LIN {X 0,Y 354.832,Z 168.283,A -85,B 0,C 180,E1 -13567.896,E2 -13567.896} C_VEL
LIN {X 0,Y 354.92,Z 168.273,A -85,B 0,C 180,E1 -13571.894,E2 -13571.894} C_VEL
LIN {X 0,Y 354.941,Z 168.271,A -85,B 0,C 180,E1 -13575.983,E2 -13575.983} C_VEL
LIN {X 0,Y 354.977,Z 168.266,A -85,B 0,C 180,E1 -13579.738,E2 -13579.738} C_VEL
LIN {X 0,Y 355.114,Z 168.252,A -85,B 0,C 180,E1 -13582.039,E2 -13582.039} C_VEL
LIN {X 0,Y 355.093,Z 168.255,A -85,B 0,C 180,E1 -13584.323,E2 -13584.323} C_VEL
LIN {X 0,Y 355.245,Z 168.235,A -85,B 0,C 180,E1 -13587.734,E2 -13587.734} C_VEL
LIN {X 0,Y 355.242,Z 168.235,A -85,B 0,C 180,E1 -13592.269,E2 -13592.269} C_VEL
LIN {X 0,Y 355.141,Z 168.245,A -85,B 0,C 180,E1 -13596.821,E2 -13596.821} C_VEL
LIN {X 0,Y 355.018,Z 168.261,A -85,B 0,C 180,E1 -13599.114,E2 -13599.114} C_VEL
LIN {X 0,Y 354.924,Z 168.271,A -85,B 0,C 180,E1 -13602.582,E2 -13602.582} C_VEL
LIN {X 0,Y 354.893,Z 168.276,A -85,B 0,C 180,E1 -13606.097,E2 -13606.097} C_VEL
LIN {X 0,Y 354.905,Z 168.274,A -85,B 0,C 180,E1 -13608.474,E2 -13608.474} C_VEL
LIN {X 0,Y 354.811,Z 168.286,A -85,B 0,C 180,E1 -13612.109,E2 -13612.109} C_VEL
LIN {X 0,Y 354.804,Z 168.287,A -85,B 0,C 180,E1 -13615.836,E2 -13615.836} C_VEL
LIN {X 0,Y 354.804,Z 168.288,A -85,B 0,C 180,E1 -13619.685,E2 -13619.685} C_VEL
LIN {X 0,Y 354.792,Z 168.29,A -85,B 0,C 180,E1 -13622.335,E2 -13622.335} C_VEL
LIN {X 0,Y 354.826,Z 168.284,A -85,B 0,C 180,E1 -13625.7,E2 -13625.7} C_VEL
LIN {X 0,Y 354.773,Z 168.291,A -85,B 0,C 180,E1 -13629.413,E2 -13629.413} C_VEL
LIN {X 0,Y 354.79,Z 168.292,A -85,B 0,C 180,E1 -13632.867,E2 -13632.867} C_VEL
LIN {X 0,Y 354.772,Z 168.293,A -85,B 0,C 180,E1 -13636.104,E2 -13636.104} C_VEL
LIN {X 0,Y 354.773,Z 168.289,A -85,B 0,C 180,E1 -13639.618,E2 -13639.618} C_VEL
LIN {X 0,Y 354.806,Z 168.29,A -85,B 0,C 180,E1 -13642.405,E2 -13642.405} C_VEL
LIN {X 0,Y 354.827,Z 168.286,A -85,B 0,C 180,E1 -13644.549,E2 -13644.549} C_VEL
LIN {X 0,Y 354.259,Z 168.738,A -85,B 0,C 180,E1 -13645.493,E2 -13645.493} C_VEL
LIN {X 0,Y 352.913,Z 169.909,A -85,B 0,C 180,E1 -13646.41,E2 -13646.41} C_VEL
LIN {X 0,Y 349.778,Z 173.519,A -85,B 0,C 180,E1 -13648.211,E2 -13648.211} C_VEL
LIN {X 0,Y 348.879,Z 176.103,A -85,B 0,C 180,E1 -13649.443,E2 -13649.443} C_VEL
LIN {X 0,Y 348.478,Z 182.428,A -85,B 0,C 180,E1 -13652.548,E2 -13652.548} C_VEL
LIN {X 0,Y 347.923,Z 189.955,A -85,B 0,C 180,E1 -13656.172,E2 -13656.172} C_VEL
LIN {X 0,Y 347.454,Z 197.78,A -85,B 0,C 180,E1 -13659.888,E2 -13659.888} C_VEL
LIN {X 0,Y 347.058,Z 205.567,A -85,B 0,C 180,E1 -13663.531,E2 -13663.531} C_VEL
LIN {X 0,Y 346.795,Z 213.332,A -85,B 0,C 180,E1 -13667.119,E2 -13667.119} C_VEL
LIN {X 0,Y 346.657,Z 216.242,A -85,B 0,C 180,E1 -13668.377,E2 -13668.377} C_VEL
LIN {X 0,Y 347.531,Z 227.151,A -85,B 0,C 180,E1 -13669.071,E2 -13669.071} C_VEL
LIN {X 0,Y 348.261,Z 236.165,A -85,B 0,C 180,E1 -13669.83,E2 -13669.83} C_VEL
LIN {X 0,Y 347.759,Z 245.798,A -85,B 0,C 180,E1 -13670.843,E2 -13670.843} C_VEL
LIN {X 0,Y 347.321,Z 255.426,A -85,B 0,C 180,E1 -13672.15,E2 -13672.15} C_VEL
LIN {X 0,Y 347.005,Z 261.907,A -85,B 0,C 180,E1 -13673.258,E2 -13673.258} C_VEL
LIN {X 0,Y 346.787,Z 268.916,A -85,B 0,C 180,E1 -13674.768,E2 -13674.768} C_VEL
LIN {X 0,Y 346.59,Z 273.17,A -85,B 0,C 180,E1 -13675.93,E2 -13675.93} C_VEL
LIN {X 0,Y 346.348,Z 277.972,A -85,B 0,C 180,E1 -13677.674,E2 -13677.674} C_VEL
LIN {X 0,Y 346.339,Z 280.246,A -85,B 0,C 180,E1 -13678.837,E2 -13678.837} C_VEL
LIN {X 0,Y 346.387,Z 281.827,A -85,B 0,C 180,E1 -13680,E2 -13680} C_VEL
LIN {X 0,Y 346.491,Z 282.748,A -85,B 0,C 180,E1 -13681.162,E2 -13681.162} C_VEL
LIN {X 0,Y 346.674,Z 283.01,A -85,B 0,C 180,E1 -13682.324,E2 -13682.324} C_VEL
LIN {X 0,Y 346.972,Z 282.623,A -85,B 0,C 180,E1 -13683.484,E2 -13683.484} C_VEL
LIN {X 0,Y 347.505,Z 281.586,A -85,B 0,C 180,E1 -13684.64,E2 -13684.64} C_VEL
LIN {X 0,Y 347.852,Z 278.872,A -85,B 0,C 180,E1 -13686.38,E2 -13686.38} C_VEL
LIN {X 0,Y 348.695,Z 274.586,A -85,B 0,C 180,E1 -13688.111,E2 -13688.111} C_VEL
LIN {X 0,Y 349.806,Z 269.133,A -85,B 0,C 180,E1 -13689.678,E2 -13689.678} C_VEL
LIN {X 0,Y 351.27,Z 261.867,A -85,B 0,C 180,E1 -13691.249,E2 -13691.249} C_VEL
LIN {X 0,Y 352.727,Z 253.419,A -85,B 0,C 180,E1 -13692.661,E2 -13692.661} C_VEL
LIN {X 0,Y 353.847,Z 246.132,A -85,B 0,C 180,E1 -13693.642,E2 -13693.642} C_VEL
LIN {X 0,Y 353.083,Z 236.877,A -85,B 0,C 180,E1 -13694.849,E2 -13694.849} C_VEL
LIN {X 0,Y 351.358,Z 227.651,A -85,B 0,C 180,E1 -13695.949,E2 -13695.949} C_VEL
LIN {X 0,Y 348.627,Z 217.69,A -85,B 0,C 180,E1 -13697.072,E2 -13697.072} C_VEL
LIN {X 0,Y 349.409,Z 211.359,A -85,B 0,C 180,E1 -13700.61,E2 -13700.61} C_VEL
LIN {X 0,Y 350.246,Z 206.213,A -85,B 0,C 180,E1 -13703.661,E2 -13703.661} C_VEL
LIN {X 0,Y 351.389,Z 200.419,A -85,B 0,C 180,E1 -13707.388,E2 -13707.388} C_VEL
LIN {X 0,Y 352.288,Z 196.86,A -85,B 0,C 180,E1 -13709.917,E2 -13709.917} C_VEL
LIN {X 0,Y 352.647,Z 195.246,A -85,B 0,C 180,E1 -13711.209,E2 -13711.209} C_VEL
LIN {X 0,Y 352.835,Z 193.025,A -85,B 0,C 180,E1 -13713.217,E2 -13713.217} C_VEL
LIN {X 0,Y 352.595,Z 190.094,A -85,B 0,C 180,E1 -13716.725,E2 -13716.725} C_VEL
LIN {X 0,Y 352.358,Z 188.51,A -85,B 0,C 180,E1 -13719.662,E2 -13719.662} C_VEL
LIN {X 0,Y 352.317,Z 187.695,A -85,B 0,C 180,E1 -13722.706,E2 -13722.706} C_VEL
LIN {X 0,Y 352.457,Z 187.837,A -85,B 0,C 180,E1 -13725.877,E2 -13725.877} C_VEL
LIN {X 0,Y 352.75,Z 188.963,A -85,B 0,C 180,E1 -13728.891,E2 -13728.891} C_VEL
LIN {X 0,Y 353.2,Z 191.093,A -85,B 0,C 180,E1 -13731.913,E2 -13731.913} C_VEL
LIN {X 0,Y 353.859,Z 194.075,A -85,B 0,C 180,E1 -13734.831,E2 -13734.831} C_VEL
LIN {X 0,Y 354.621,Z 197.872,A -85,B 0,C 180,E1 -13737.648,E2 -13737.648} C_VEL
LIN {X 0,Y 355.095,Z 201.146,A -85,B 0,C 180,E1 -13739.687,E2 -13739.687} C_VEL
LIN {X 0,Y 354.861,Z 203.838,A -85,B 0,C 180,E1 -13741.084,E2 -13741.084} C_VEL
LIN {X 0,Y 352.926,Z 210.525,A -85,B 0,C 180,E1 -13744.016,E2 -13744.016} C_VEL
LIN {X 0,Y 350.745,Z 220.327,A -85,B 0,C 180,E1 -13747.931,E2 -13747.931} C_VEL
LIN {X 0,Y 353.911,Z 233.578,A -85,B 0,C 180,E1 -13748.961,E2 -13748.961} C_VEL
LIN {X 0,Y 355.2,Z 243.511,A -85,B 0,C 180,E1 -13749.771,E2 -13749.771} C_VEL
LIN {X 0,Y 355.188,Z 251.982,A -85,B 0,C 180,E1 -13750.493,E2 -13750.493} C_VEL
LIN {X 0,Y 353.684,Z 263.835,A -85,B 0,C 180,E1 -13751.61,E2 -13751.61} C_VEL
LIN {X 0,Y 352.068,Z 274.487,A -85,B 0,C 180,E1 -13752.874,E2 -13752.874} C_VEL
LIN {X 0,Y 350.347,Z 284.861,A -85,B 0,C 180,E1 -13754.429,E2 -13754.429} C_VEL
LIN {X 0,Y 349.222,Z 293.327,A -85,B 0,C 180,E1 -13756.023,E2 -13756.023} C_VEL
LIN {X 0,Y 348.027,Z 300.772,A -85,B 0,C 180,E1 -13757.757,E2 -13757.757} C_VEL
LIN {X 0,Y 347.198,Z 306.772,A -85,B 0,C 180,E1 -13759.502,E2 -13759.502} C_VEL
LIN {X 0,Y 346.647,Z 311.533,A -85,B 0,C 180,E1 -13761.252,E2 -13761.252} C_VEL
LIN {X 0,Y 346.342,Z 315.161,A -85,B 0,C 180,E1 -13763.005,E2 -13763.005} C_VEL
LIN {X 0,Y 346.251,Z 316.986,A -85,B 0,C 180,E1 -13764.173,E2 -13764.173} C_VEL
LIN {X 0,Y 346.215,Z 318.385,A -85,B 0,C 180,E1 -13765.341,E2 -13765.341} C_VEL
LIN {X 0,Y 346.197,Z 319.375,A -85,B 0,C 180,E1 -13766.507,E2 -13766.507} C_VEL
LIN {X 0,Y 346.245,Z 319.9,A -85,B 0,C 180,E1 -13767.672,E2 -13767.672} C_VEL
LIN {X 0,Y 346.385,Z 320.016,A -85,B 0,C 180,E1 -13768.836,E2 -13768.836} C_VEL
LIN {X 0,Y 346.394,Z 319.713,A -85,B 0,C 180,E1 -13769.998,E2 -13769.998} C_VEL
LIN {X 0,Y 346.419,Z 318.933,A -85,B 0,C 180,E1 -13771.161,E2 -13771.161} C_VEL
LIN {X 0,Y 346.459,Z 317.723,A -85,B 0,C 180,E1 -13772.323,E2 -13772.323} C_VEL
LIN {X 0,Y 346.313,Z 315.011,A -85,B 0,C 180,E1 -13774.071,E2 -13774.071} C_VEL
LIN {X 0,Y 346.396,Z 311.191,A -85,B 0,C 180,E1 -13775.82,E2 -13775.82} C_VEL
LIN {X 0,Y 346.496,Z 306.1,A -85,B 0,C 180,E1 -13777.574,E2 -13777.574} C_VEL
LIN {X 0,Y 346.692,Z 299.54,A -85,B 0,C 180,E1 -13779.331,E2 -13779.331} C_VEL
LIN {X 0,Y 347.11,Z 291.289,A -85,B 0,C 180,E1 -13781.088,E2 -13781.088} C_VEL
LIN {X 0,Y 347.617,Z 282.661,A -85,B 0,C 180,E1 -13782.551,E2 -13782.551} C_VEL
LIN {X 0,Y 348.249,Z 273.162,A -85,B 0,C 180,E1 -13783.864,E2 -13783.864} C_VEL
LIN {X 0,Y 348.924,Z 262.248,A -85,B 0,C 180,E1 -13785.073,E2 -13785.073} C_VEL
LIN {X 0,Y 349.637,Z 251.072,A -85,B 0,C 180,E1 -13786.043,E2 -13786.043} C_VEL
LIN {X 0,Y 349.783,Z 243.763,A -85,B 0,C 180,E1 -13786.56,E2 -13786.56} C_VEL
LIN {X 0,Y 348.453,Z 230.087,A -85,B 0,C 180,E1 -13787.324,E2 -13787.324} C_VEL
LIN {X 0,Y 347.768,Z 220.166,A -85,B 0,C 180,E1 -13787.729,E2 -13787.729} C_VEL
LIN {X 0,Y 349.042,Z 206.707,A -85,B 0,C 180,E1 -13792.147,E2 -13792.147} C_VEL
LIN {X 0,Y 350.509,Z 194.632,A -85,B 0,C 180,E1 -13796.173,E2 -13796.173} C_VEL
LIN {X 0,Y 351.264,Z 188.272,A -85,B 0,C 180,E1 -13798.316,E2 -13798.316} C_VEL
LIN {X 0,Y 350.363,Z 182.502,A -85,B 0,C 180,E1 -13800.396,E2 -13800.396} C_VEL
LIN {X 0,Y 348.285,Z 171.813,A -85,B 0,C 180,E1 -13804.4,E2 -13804.4} C_VEL
LIN {X 0,Y 347.78,Z 169.17,A -85,B 0,C 180,E1 -13805.428,E2 -13805.428} C_VEL
LIN {X 0,Y 347.745,Z 169.171,A -85,B 0,C 180,E1 -13808.791,E2 -13808.791} C_VEL
LIN {X 0,Y 347.742,Z 169.166,A -85,B 0,C 180,E1 -13811.828,E2 -13811.828} C_VEL
LIN {X 0,Y 347.789,Z 169.162,A -85,B 0,C 180,E1 -13815.01,E2 -13815.01} C_VEL
LIN {X 0,Y 347.775,Z 169.167,A -85,B 0,C 180,E1 -13818.389,E2 -13818.389} C_VEL
LIN {X 0,Y 347.767,Z 169.167,A -85,B 0,C 180,E1 -13822.009,E2 -13822.009} C_VEL
LIN {X 0,Y 347.733,Z 169.168,A -85,B 0,C 180,E1 -13825.535,E2 -13825.535} C_VEL
LIN {X 0,Y 347.752,Z 169.168,A -85,B 0,C 180,E1 -13829.652,E2 -13829.652} C_VEL
LIN {X 0,Y 347.84,Z 169.154,A -85,B 0,C 180,E1 -13832.743,E2 -13832.743} C_VEL
LIN {X 0,Y 347.772,Z 169.165,A -85,B 0,C 180,E1 -13836.161,E2 -13836.161} C_VEL
LIN {X 0,Y 347.798,Z 169.163,A -85,B 0,C 180,E1 -13839.908,E2 -13839.908} C_VEL
LIN {X 0,Y 347.853,Z 169.153,A -85,B 0,C 180,E1 -13842.358,E2 -13842.358} C_VEL
LIN {X 0,Y 347.883,Z 169.15,A -85,B 0,C 180,E1 -13845.97,E2 -13845.97} C_VEL
LIN {X 0,Y 347.916,Z 169.148,A -85,B 0,C 180,E1 -13849.525,E2 -13849.525} C_VEL
LIN {X 0,Y 348.081,Z 169.128,A -85,B 0,C 180,E1 -13853.042,E2 -13853.042} C_VEL
LIN {X 0,Y 348.195,Z 169.111,A -85,B 0,C 180,E1 -13857.686,E2 -13857.686} C_VEL
LIN {X 0,Y 348.331,Z 169.093,A -85,B 0,C 180,E1 -13860,E2 -13860} C_VEL
LIN {X 0,Y 348.189,Z 169.111,A -85,B 0,C 180,E1 -13862.314,E2 -13862.314} C_VEL
LIN {X 0,Y 348.091,Z 169.127,A -85,B 0,C 180,E1 -13866.958,E2 -13866.958} C_VEL
LIN {X 0,Y 347.955,Z 169.141,A -85,B 0,C 180,E1 -13869.299,E2 -13869.299} C_VEL
LIN {X 0,Y 347.88,Z 169.152,A -85,B 0,C 180,E1 -13872.84,E2 -13872.84} C_VEL
LIN {X 0,Y 347.826,Z 169.161,A -85,B 0,C 180,E1 -13876.432,E2 -13876.432} C_VEL
LIN {X 0,Y 347.846,Z 169.155,A -85,B 0,C 180,E1 -13878.861,E2 -13878.861} C_VEL
LIN {X 0,Y 347.768,Z 169.166,A -85,B 0,C 180,E1 -13882.58,E2 -13882.58} C_VEL
LIN {X 0,Y 347.774,Z 169.162,A -85,B 0,C 180,E1 -13885.111,E2 -13885.111} C_VEL
LIN {X 0,Y 347.733,Z 169.167,A -85,B 0,C 180,E1 -13889.016,E2 -13889.016} C_VEL
LIN {X 0,Y 347.726,Z 169.173,A -85,B 0,C 180,E1 -13891.915,E2 -13891.915} C_VEL
LIN {X 0,Y 347.778,Z 169.167,A -85,B 0,C 180,E1 -13895.877,E2 -13895.877} C_VEL
LIN {X 0,Y 347.742,Z 169.166,A -85,B 0,C 180,E1 -13898.794,E2 -13898.794} C_VEL
LIN {X 0,Y 347.741,Z 169.17,A -85,B 0,C 180,E1 -13901.832,E2 -13901.832} C_VEL
LIN {X 0,Y 347.757,Z 169.166,A -85,B 0,C 180,E1 -13905.018,E2 -13905.018} C_VEL
LIN {X 0,Y 347.741,Z 169.166,A -85,B 0,C 180,E1 -13908.399,E2 -13908.399} C_VEL
LIN {X 0,Y 347.765,Z 169.163,A -85,B 0,C 180,E1 -13912.013,E2 -13912.013} C_VEL
LIN {X 0,Y 347.737,Z 169.169,A -85,B 0,C 180,E1 -13915.538,E2 -13915.538} C_VEL
LIN {X 0,Y 347.759,Z 169.165,A -85,B 0,C 180,E1 -13919.656,E2 -13919.656} C_VEL
LIN {X 0,Y 347.847,Z 169.157,A -85,B 0,C 180,E1 -13922.746,E2 -13922.746} C_VEL
LIN {X 0,Y 347.784,Z 169.161,A -85,B 0,C 180,E1 -13926.164,E2 -13926.164} C_VEL
LIN {X 0,Y 347.81,Z 169.158,A -85,B 0,C 180,E1 -13929.911,E2 -13929.911} C_VEL
LIN {X 0,Y 347.864,Z 169.155,A -85,B 0,C 180,E1 -13932.361,E2 -13932.361} C_VEL
LIN {X 0,Y 347.896,Z 169.149,A -85,B 0,C 180,E1 -13935.973,E2 -13935.973} C_VEL
LIN {X 0,Y 347.927,Z 169.143,A -85,B 0,C 180,E1 -13939.528,E2 -13939.528} C_VEL
LIN {X 0,Y 348.075,Z 169.127,A -85,B 0,C 180,E1 -13941.877,E2 -13941.877} C_VEL
LIN {X 0,Y 348.068,Z 169.13,A -85,B 0,C 180,E1 -13944.208,E2 -13944.208} C_VEL
LIN {X 0,Y 348.207,Z 169.111,A -85,B 0,C 180,E1 -13947.688,E2 -13947.688} C_VEL
LIN {X 0,Y 348.119,Z 169.119,A -85,B 0,C 180,E1 -13951.159,E2 -13951.159} C_VEL
LIN {X 0,Y 348.204,Z 169.111,A -85,B 0,C 180,E1 -13952.315,E2 -13952.315} C_VEL
LIN {X 0,Y 348.109,Z 169.121,A -85,B 0,C 180,E1 -13956.959,E2 -13956.959} C_VEL
LIN {X 0,Y 347.971,Z 169.14,A -85,B 0,C 180,E1 -13959.3,E2 -13959.3} C_VEL
LIN {X 0,Y 347.893,Z 169.148,A -85,B 0,C 180,E1 -13962.841,E2 -13962.841} C_VEL
LIN {X 0,Y 347.843,Z 169.154,A -85,B 0,C 180,E1 -13966.433,E2 -13966.433} C_VEL
LIN {X 0,Y 347.855,Z 169.154,A -85,B 0,C 180,E1 -13968.862,E2 -13968.862} C_VEL
LIN {X 0,Y 347.753,Z 169.166,A -85,B 0,C 180,E1 -13972.582,E2 -13972.582} C_VEL
LIN {X 0,Y 347.741,Z 169.171,A -85,B 0,C 180,E1 -13975.116,E2 -13975.116} C_VEL
LIN {X 0,Y 347.733,Z 169.168,A -85,B 0,C 180,E1 -13977.702,E2 -13977.702} C_VEL
LIN {X 0,Y 347.745,Z 169.167,A -85,B 0,C 180,E1 -13980.35,E2 -13980.35} C_VEL
LIN {X 0,Y 347.753,Z 169.165,A -85,B 0,C 180,E1 -13984.045,E2 -13984.045} C_VEL
LIN {X 0,Y 347.761,Z 169.165,A -85,B 0,C 180,E1 -13987.323,E2 -13987.323} C_VEL
LIN {X 0,Y 347.746,Z 169.166,A -85,B 0,C 180,E1 -13991.602,E2 -13991.602} C_VEL
LIN {X 0,Y 347.71,Z 169.172,A -85,B 0,C 180,E1 -13995.028,E2 -13995.028} C_VEL
LIN {X 0,Y 347.755,Z 169.17,A -85,B 0,C 180,E1 -13998.398,E2 -13998.398} C_VEL
LIN {X 0,Y 347.769,Z 169.166,A -85,B 0,C 180,E1 -14002.014,E2 -14002.014} C_VEL
LIN {X 0,Y 347.891,Z 169.301,A -85,B 0,C 180,E1 -14005.924,E2 -14005.924} C_VEL
LIN {X 0,Y 348.865,Z 175.399,A -85,B 0,C 180,E1 -14009.089,E2 -14009.089} C_VEL
LIN {X 0,Y 348.879,Z 176.103,A -85,B 0,C 180,E1 -14009.443,E2 -14009.443} C_VEL
LIN {X 0,Y 348.575,Z 177.366,A -85,B 0,C 180,E1 -14010.052,E2 -14010.052} C_VEL
LIN {X 0,Y 347.164,Z 179.348,A -85,B 0,C 180,E1 -14010.942,E2 -14010.942} C_VEL
LIN {X 0,Y 342.5,Z 184.068,A -85,B 0,C 180,E1 -14012.987,E2 -14012.987} C_VEL
LIN {X 0,Y 341.299,Z 186.067,A -85,B 0,C 180,E1 -14013.908,E2 -14013.908} C_VEL
LIN {X 0,Y 341.173,Z 186.718,A -85,B 0,C 180,E1 -14014.223,E2 -14014.223} C_VEL
LIN {X 0,Y 340.593,Z 194.922,A -85,B 0,C 180,E1 -14018.214,E2 -14018.214} C_VEL
LIN {X 0,Y 340.171,Z 202.705,A -85,B 0,C 180,E1 -14021.947,E2 -14021.947} C_VEL
LIN {X 0,Y 339.795,Z 210.51,A -85,B 0,C 180,E1 -14025.629,E2 -14025.629} C_VEL
LIN {X 0,Y 339.588,Z 216.104,A -85,B 0,C 180,E1 -14028.245,E2 -14028.245} C_VEL
LIN {X 0,Y 340.465,Z 227.524,A -85,B 0,C 180,E1 -14028.992,E2 -14028.992} C_VEL
LIN {X 0,Y 341.174,Z 236.474,A -85,B 0,C 180,E1 -14029.766,E2 -14029.766} C_VEL
LIN {X 0,Y 340.678,Z 246.059,A -85,B 0,C 180,E1 -14030.8,E2 -14030.8} C_VEL
LIN {X 0,Y 340.261,Z 254.913,A -85,B 0,C 180,E1 -14032.016,E2 -14032.016} C_VEL
LIN {X 0,Y 339.898,Z 262.342,A -85,B 0,C 180,E1 -14033.302,E2 -14033.302} C_VEL
LIN {X 0,Y 339.715,Z 268.591,A -85,B 0,C 180,E1 -14034.658,E2 -14034.658} C_VEL
LIN {X 0,Y 339.517,Z 272.979,A -85,B 0,C 180,E1 -14035.845,E2 -14035.845} C_VEL
LIN {X 0,Y 339.256,Z 277.973,A -85,B 0,C 180,E1 -14037.626,E2 -14037.626} C_VEL
LIN {X 0,Y 339.241,Z 280.36,A -85,B 0,C 180,E1 -14038.813,E2 -14038.813} C_VEL
LIN {X 0,Y 339.291,Z 282.052,A -85,B 0,C 180,E1 -14040,E2 -14040} C_VEL
LIN {X 0,Y 339.412,Z 283.079,A -85,B 0,C 180,E1 -14041.187,E2 -14041.187} C_VEL
LIN {X 0,Y 339.619,Z 283.463,A -85,B 0,C 180,E1 -14042.372,E2 -14042.372} C_VEL
LIN {X 0,Y 339.928,Z 283.206,A -85,B 0,C 180,E1 -14043.556,E2 -14043.556} C_VEL
LIN {X 0,Y 340.484,Z 282.3,A -85,B 0,C 180,E1 -14044.736,E2 -14044.736} C_VEL
LIN {X 0,Y 340.876,Z 279.802,A -85,B 0,C 180,E1 -14046.511,E2 -14046.511} C_VEL
LIN {X 0,Y 341.78,Z 275.746,A -85,B 0,C 180,E1 -14048.276,E2 -14048.276} C_VEL
LIN {X 0,Y 342.955,Z 270.549,A -85,B 0,C 180,E1 -14049.873,E2 -14049.873} C_VEL
LIN {X 0,Y 344.463,Z 263.633,A -85,B 0,C 180,E1 -14051.474,E2 -14051.474} C_VEL
LIN {X 0,Y 345.996,Z 255.595,A -85,B 0,C 180,E1 -14052.911,E2 -14052.911} C_VEL
LIN {X 0,Y 347.357,Z 247.616,A -85,B 0,C 180,E1 -14054.052,E2 -14054.052} C_VEL
LIN {X 0,Y 346.598,Z 237.738,A -85,B 0,C 180,E1 -14055.413,E2 -14055.413} C_VEL
LIN {X 0,Y 344.576,Z 227.433,A -85,B 0,C 180,E1 -14056.715,E2 -14056.715} C_VEL
LIN {X 0,Y 341.877,Z 217.803,A -85,B 0,C 180,E1 -14057.875,E2 -14057.875} C_VEL
LIN {X 0,Y 342.757,Z 211.316,A -85,B 0,C 180,E1 -14061.659,E2 -14061.659} C_VEL
LIN {X 0,Y 343.884,Z 205.368,A -85,B 0,C 180,E1 -14065.416,E2 -14065.416} C_VEL
LIN {X 0,Y 345.235,Z 199.882,A -85,B 0,C 180,E1 -14069.247,E2 -14069.247} C_VEL
LIN {X 0,Y 345.94,Z 196.683,A -85,B 0,C 180,E1 -14071.885,E2 -14071.885} C_VEL
LIN {X 0,Y 346.074,Z 194.913,A -85,B 0,C 180,E1 -14073.629,E2 -14073.629} C_VEL
LIN {X 0,Y 345.922,Z 192.947,A -85,B 0,C 180,E1 -14076.099,E2 -14076.099} C_VEL
LIN {X 0,Y 345.726,Z 191.097,A -85,B 0,C 180,E1 -14079.422,E2 -14079.422} C_VEL
LIN {X 0,Y 345.691,Z 190.303,A -85,B 0,C 180,E1 -14082.137,E2 -14082.137} C_VEL
LIN {X 0,Y 345.78,Z 190.316,A -85,B 0,C 180,E1 -14085.347,E2 -14085.347} C_VEL
LIN {X 0,Y 346.119,Z 191.449,A -85,B 0,C 180,E1 -14088.703,E2 -14088.703} C_VEL
LIN {X 0,Y 346.448,Z 192.947,A -85,B 0,C 180,E1 -14091.032,E2 -14091.032} C_VEL
LIN {X 0,Y 347.012,Z 195.799,A -85,B 0,C 180,E1 -14094.108,E2 -14094.108} C_VEL
LIN {X 0,Y 347.713,Z 199.217,A -85,B 0,C 180,E1 -14096.924,E2 -14096.924} C_VEL
LIN {X 0,Y 348.356,Z 203.497,A -85,B 0,C 180,E1 -14099.709,E2 -14099.709} C_VEL
LIN {X 0,Y 348.047,Z 205.947,A -85,B 0,C 180,E1 -14101.011,E2 -14101.011} C_VEL
LIN {X 0,Y 345.944,Z 212.854,A -85,B 0,C 180,E1 -14104.1,E2 -14104.1} C_VEL
LIN {X 0,Y 344.188,Z 220.498,A -85,B 0,C 180,E1 -14107.214,E2 -14107.214} C_VEL
LIN {X 0,Y 347.3,Z 233.012,A -85,B 0,C 180,E1 -14108.247,E2 -14108.247} C_VEL
LIN {X 0,Y 348.727,Z 242.947,A -85,B 0,C 180,E1 -14109.109,E2 -14109.109} C_VEL
LIN {X 0,Y 348.94,Z 250.902,A -85,B 0,C 180,E1 -14109.83,E2 -14109.83} C_VEL
LIN {X 0,Y 347.641,Z 261.448,A -85,B 0,C 180,E1 -14110.82,E2 -14110.82} C_VEL
LIN {X 0,Y 345.878,Z 272.374,A -85,B 0,C 180,E1 -14112.1,E2 -14112.1} C_VEL
LIN {X 0,Y 344.343,Z 281.345,A -85,B 0,C 180,E1 -14113.395,E2 -14113.395} C_VEL
LIN {X 0,Y 342.912,Z 289.582,A -85,B 0,C 180,E1 -14114.85,E2 -14114.85} C_VEL
LIN {X 0,Y 341.712,Z 297.635,A -85,B 0,C 180,E1 -14116.62,E2 -14116.62} C_VEL
LIN {X 0,Y 340.673,Z 303.161,A -85,B 0,C 180,E1 -14118.093,E2 -14118.093} C_VEL
LIN {X 0,Y 339.97,Z 308.573,A -85,B 0,C 180,E1 -14119.878,E2 -14119.878} C_VEL
LIN {X 0,Y 339.49,Z 312.803,A -85,B 0,C 180,E1 -14121.666,E2 -14121.666} C_VEL
LIN {X 0,Y 339.27,Z 315.025,A -85,B 0,C 180,E1 -14122.858,E2 -14122.858} C_VEL
LIN {X 0,Y 339.172,Z 316.779,A -85,B 0,C 180,E1 -14124.051,E2 -14124.051} C_VEL
LIN {X 0,Y 339.116,Z 318.124,A -85,B 0,C 180,E1 -14125.243,E2 -14125.243} C_VEL
LIN {X 0,Y 339.118,Z 319.022,A -85,B 0,C 180,E1 -14126.434,E2 -14126.434} C_VEL
LIN {X 0,Y 339.32,Z 319.554,A -85,B 0,C 180,E1 -14128.811,E2 -14128.811} C_VEL
LIN {X 0,Y 339.333,Z 319.161,A -85,B 0,C 180,E1 -14129.998,E2 -14129.998} C_VEL
LIN {X 0,Y 339.359,Z 318.32,A -85,B 0,C 180,E1 -14131.185,E2 -14131.185} C_VEL
LIN {X 0,Y 339.377,Z 317.058,A -85,B 0,C 180,E1 -14132.372,E2 -14132.372} C_VEL
LIN {X 0,Y 339.248,Z 314.236,A -85,B 0,C 180,E1 -14134.156,E2 -14134.156} C_VEL
LIN {X 0,Y 339.346,Z 310.271,A -85,B 0,C 180,E1 -14135.942,E2 -14135.942} C_VEL
LIN {X 0,Y 339.504,Z 304.01,A -85,B 0,C 180,E1 -14138.03,E2 -14138.03} C_VEL
LIN {X 0,Y 339.748,Z 297.01,A -85,B 0,C 180,E1 -14139.824,E2 -14139.824} C_VEL
LIN {X 0,Y 340.251,Z 288.161,A -85,B 0,C 180,E1 -14141.616,E2 -14141.616} C_VEL
LIN {X 0,Y 340.79,Z 278.903,A -85,B 0,C 180,E1 -14143.11,E2 -14143.11} C_VEL
LIN {X 0,Y 341.326,Z 269.819,A -85,B 0,C 180,E1 -14144.303,E2 -14144.303} C_VEL
LIN {X 0,Y 342.159,Z 258.675,A -85,B 0,C 180,E1 -14145.485,E2 -14145.485} C_VEL
LIN {X 0,Y 342.768,Z 246.853,A -85,B 0,C 180,E1 -14146.45,E2 -14146.45} C_VEL
LIN {X 0,Y 342.108,Z 238.206,A -85,B 0,C 180,E1 -14147.02,E2 -14147.02} C_VEL
LIN {X 0,Y 340.969,Z 224.813,A -85,B 0,C 180,E1 -14147.678,E2 -14147.678} C_VEL
LIN {X 0,Y 340.716,Z 220.142,A -85,B 0,C 180,E1 -14147.866,E2 -14147.866} C_VEL
LIN {X 0,Y 342.045,Z 206.743,A -85,B 0,C 180,E1 -14152.389,E2 -14152.389} C_VEL
LIN {X 0,Y 343.429,Z 195.681,A -85,B 0,C 180,E1 -14156.166,E2 -14156.166} C_VEL
LIN {X 0,Y 344.177,Z 190.335,A -85,B 0,C 180,E1 -14158.009,E2 -14158.009} C_VEL
LIN {X 0,Y 343.936,Z 186.546,A -85,B 0,C 180,E1 -14159.365,E2 -14159.365} C_VEL
LIN {X 0,Y 341.942,Z 176.601,A -85,B 0,C 180,E1 -14163.117,E2 -14163.117} C_VEL
LIN {X 0,Y 340.76,Z 170.046,A -85,B 0,C 180,E1 -14165.725,E2 -14165.725} C_VEL
LIN {X 0,Y 340.702,Z 170.046,A -85,B 0,C 180,E1 -14168.384,E2 -14168.384} C_VEL
LIN {X 0,Y 340.691,Z 170.045,A -85,B 0,C 180,E1 -14172.044,E2 -14172.044} C_VEL
LIN {X 0,Y 340.713,Z 170.042,A -85,B 0,C 180,E1 -14175.466,E2 -14175.466} C_VEL
LIN {X 0,Y 340.716,Z 170.044,A -85,B 0,C 180,E1 -14178.695,E2 -14178.695} C_VEL
LIN {X 0,Y 340.727,Z 170.041,A -85,B 0,C 180,E1 -14181.772,E2 -14181.772} C_VEL
LIN {X 0,Y 340.711,Z 170.043,A -85,B 0,C 180,E1 -14185.594,E2 -14185.594} C_VEL
LIN {X 0,Y 340.692,Z 170.044,A -85,B 0,C 180,E1 -14188.955,E2 -14188.955} C_VEL
LIN {X 0,Y 340.767,Z 170.036,A -85,B 0,C 180,E1 -14192.473,E2 -14192.473} C_VEL
LIN {X 0,Y 340.741,Z 170.042,A -85,B 0,C 180,E1 -14195.637,E2 -14195.637} C_VEL
LIN {X 0,Y 340.724,Z 170.044,A -85,B 0,C 180,E1 -14199.473,E2 -14199.473} C_VEL
LIN {X 0,Y 340.845,Z 170.028,A -85,B 0,C 180,E1 -14201.983,E2 -14201.983} C_VEL
LIN {X 0,Y 340.855,Z 170.028,A -85,B 0,C 180,E1 -14205.704,E2 -14205.704} C_VEL
LIN {X 0,Y 340.859,Z 170.028,A -85,B 0,C 180,E1 -14209.306,E2 -14209.306} C_VEL
LIN {X 0,Y 341.048,Z 170.002,A -85,B 0,C 180,E1 -14212.898,E2 -14212.898} C_VEL
LIN {X 0,Y 341.157,Z 169.988,A -85,B 0,C 180,E1 -14217.639,E2 -14217.639} C_VEL
LIN {X 0,Y 341.281,Z 169.971,A -85,B 0,C 180,E1 -14220,E2 -14220} C_VEL
LIN {X 0,Y 341.151,Z 169.988,A -85,B 0,C 180,E1 -14222.361,E2 -14222.361} C_VEL
LIN {X 0,Y 341.061,Z 170.001,A -85,B 0,C 180,E1 -14227.102,E2 -14227.102} C_VEL
LIN {X 0,Y 340.861,Z 170.028,A -85,B 0,C 180,E1 -14230.694,E2 -14230.694} C_VEL
LIN {X 0,Y 340.849,Z 170.029,A -85,B 0,C 180,E1 -14234.325,E2 -14234.325} C_VEL
LIN {X 0,Y 340.825,Z 170.032,A -85,B 0,C 180,E1 -14238.468,E2 -14238.468} C_VEL
LIN {X 0,Y 340.74,Z 170.04,A -85,B 0,C 180,E1 -14241.858,E2 -14241.858} C_VEL
LIN {X 0,Y 340.724,Z 170.042,A -85,B 0,C 180,E1 -14245.668,E2 -14245.668} C_VEL
LIN {X 0,Y 340.695,Z 170.046,A -85,B 0,C 180,E1 -14249.675,E2 -14249.675} C_VEL
LIN {X 0,Y 340.674,Z 170.048,A -85,B 0,C 180,E1 -14252.437,E2 -14252.437} C_VEL
LIN {X 0,Y 340.707,Z 170.044,A -85,B 0,C 180,E1 -14255.28,E2 -14255.28} C_VEL
LIN {X 0,Y 340.701,Z 170.044,A -85,B 0,C 180,E1 -14258.388,E2 -14258.388} C_VEL
LIN {X 0,Y 340.689,Z 170.046,A -85,B 0,C 180,E1 -14262.047,E2 -14262.047} C_VEL
LIN {X 0,Y 340.675,Z 170.051,A -85,B 0,C 180,E1 -14265.463,E2 -14265.463} C_VEL
LIN {X 0,Y 340.677,Z 170.047,A -85,B 0,C 180,E1 -14268.692,E2 -14268.692} C_VEL
LIN {X 0,Y 340.724,Z 170.042,A -85,B 0,C 180,E1 -14271.774,E2 -14271.774} C_VEL
LIN {X 0,Y 340.716,Z 170.043,A -85,B 0,C 180,E1 -14275.597,E2 -14275.597} C_VEL
LIN {X 0,Y 340.698,Z 170.049,A -85,B 0,C 180,E1 -14278.958,E2 -14278.958} C_VEL
LIN {X 0,Y 340.775,Z 170.036,A -85,B 0,C 180,E1 -14282.476,E2 -14282.476} C_VEL
LIN {X 0,Y 340.751,Z 170.037,A -85,B 0,C 180,E1 -14285.64,E2 -14285.64} C_VEL
LIN {X 0,Y 340.75,Z 170.037,A -85,B 0,C 180,E1 -14289.477,E2 -14289.477} C_VEL
LIN {X 0,Y 340.855,Z 170.025,A -85,B 0,C 180,E1 -14291.986,E2 -14291.986} C_VEL
LIN {X 0,Y 340.867,Z 170.023,A -85,B 0,C 180,E1 -14295.707,E2 -14295.707} C_VEL
LIN {X 0,Y 340.87,Z 170.022,A -85,B 0,C 180,E1 -14299.308,E2 -14299.308} C_VEL
LIN {X 0,Y 341.076,Z 169.997,A -85,B 0,C 180,E1 -14302.9,E2 -14302.9} C_VEL
LIN {X 0,Y 341.169,Z 169.987,A -85,B 0,C 180,E1 -14307.641,E2 -14307.641} C_VEL
LIN {X 0,Y 341.09,Z 169.995,A -85,B 0,C 180,E1 -14311.182,E2 -14311.182} C_VEL
LIN {X 0,Y 341.166,Z 169.987,A -85,B 0,C 180,E1 -14312.363,E2 -14312.363} C_VEL
LIN {X 0,Y 341.079,Z 169.997,A -85,B 0,C 180,E1 -14317.103,E2 -14317.103} C_VEL
LIN {X 0,Y 340.874,Z 170.022,A -85,B 0,C 180,E1 -14320.695,E2 -14320.695} C_VEL
LIN {X 0,Y 340.867,Z 170.023,A -85,B 0,C 180,E1 -14324.326,E2 -14324.326} C_VEL
LIN {X 0,Y 340.841,Z 170.026,A -85,B 0,C 180,E1 -14328.468,E2 -14328.468} C_VEL
LIN {X 0,Y 340.722,Z 170.042,A -85,B 0,C 180,E1 -14331.843,E2 -14331.843} C_VEL
LIN {X 0,Y 340.674,Z 170.047,A -85,B 0,C 180,E1 -14335.674,E2 -14335.674} C_VEL
LIN {X 0,Y 340.683,Z 170.046,A -85,B 0,C 180,E1 -14338.327,E2 -14338.327} C_VEL
LIN {X 0,Y 340.699,Z 170.048,A -85,B 0,C 180,E1 -14341.046,E2 -14341.046} C_VEL
LIN {X 0,Y 340.722,Z 170.042,A -85,B 0,C 180,E1 -14345.28,E2 -14345.28} C_VEL
LIN {X 0,Y 340.698,Z 170.046,A -85,B 0,C 180,E1 -14348.383,E2 -14348.383} C_VEL
LIN {X 0,Y 340.698,Z 170.045,A -85,B 0,C 180,E1 -14352.045,E2 -14352.045} C_VEL
LIN {X 0,Y 340.657,Z 170.052,A -85,B 0,C 180,E1 -14356.228,E2 -14356.228} C_VEL
LIN {X 0,Y 340.682,Z 170.046,A -85,B 0,C 180,E1 -14359.756,E2 -14359.756} C_VEL
LIN {X 0,Y 340.709,Z 170.042,A -85,B 0,C 180,E1 -14363.259,E2 -14363.259} C_VEL
LIN {X 0,Y 340.84,Z 170.119,A -85,B 0,C 180,E1 -14365.779,E2 -14365.779} C_VEL
LIN {X 0,Y 341.847,Z 176.362,A -85,B 0,C 180,E1 -14369.071,E2 -14369.071} C_VEL
LIN {X 0,Y 341.483,Z 182.722,A -85,B 0,C 180,E1 -14372.251,E2 -14372.251} C_VEL
LIN {X 0,Y 341.173,Z 186.718,A -85,B 0,C 180,E1 -14374.223,E2 -14374.223} C_VEL
LIN {X 0,Y 340.384,Z 188.684,A -85,B 0,C 180,E1 -14375.149,E2 -14375.149} C_VEL
LIN {X 0,Y 337.305,Z 192.041,A -85,B 0,C 180,E1 -14376.638,E2 -14376.638} C_VEL
LIN {X 0,Y 334.698,Z 194.736,A -85,B 0,C 180,E1 -14377.843,E2 -14377.843} C_VEL
LIN {X 0,Y 333.524,Z 196.748,A -85,B 0,C 180,E1 -14378.783,E2 -14378.783} C_VEL
LIN {X 0,Y 333.397,Z 197.411,A -85,B 0,C 180,E1 -14379.103,E2 -14379.103} C_VEL
LIN {X 0,Y 332.987,Z 205.043,A -85,B 0,C 180,E1 -14382.814,E2 -14382.814} C_VEL
LIN {X 0,Y 332.655,Z 212.876,A -85,B 0,C 180,E1 -14386.562,E2 -14386.562} C_VEL
LIN {X 0,Y 332.539,Z 216.296,A -85,B 0,C 180,E1 -14388.147,E2 -14388.147} C_VEL
LIN {X 0,Y 333.349,Z 227.692,A -85,B 0,C 180,E1 -14388.908,E2 -14388.908} C_VEL
LIN {X 0,Y 334.096,Z 236.643,A -85,B 0,C 180,E1 -14389.7,E2 -14389.7} C_VEL
LIN {X 0,Y 333.598,Z 246.242,A -85,B 0,C 180,E1 -14390.756,E2 -14390.756} C_VEL
LIN {X 0,Y 333.147,Z 255.87,A -85,B 0,C 180,E1 -14392.119,E2 -14392.119} C_VEL
LIN {X 0,Y 332.758,Z 264.18,A -85,B 0,C 180,E1 -14393.642,E2 -14393.642} C_VEL
LIN {X 0,Y 332.566,Z 270.59,A -85,B 0,C 180,E1 -14395.151,E2 -14395.151} C_VEL
LIN {X 0,Y 332.253,Z 276.392,A -85,B 0,C 180,E1 -14396.969,E2 -14396.969} C_VEL
LIN {X 0,Y 332.143,Z 280.427,A -85,B 0,C 180,E1 -14398.788,E2 -14398.788} C_VEL
LIN {X 0,Y 332.194,Z 282.244,A -85,B 0,C 180,E1 -14400,E2 -14400} C_VEL
LIN {X 0,Y 332.335,Z 283.402,A -85,B 0,C 180,E1 -14401.212,E2 -14401.212} C_VEL
LIN {X 0,Y 332.566,Z 283.918,A -85,B 0,C 180,E1 -14402.422,E2 -14402.422} C_VEL
LIN {X 0,Y 332.885,Z 283.791,A -85,B 0,C 180,E1 -14403.631,E2 -14403.631} C_VEL
LIN {X 0,Y 333.447,Z 283.004,A -85,B 0,C 180,E1 -14404.836,E2 -14404.836} C_VEL
LIN {X 0,Y 333.882,Z 280.703,A -85,B 0,C 180,E1 -14406.648,E2 -14406.648} C_VEL
LIN {X 0,Y 334.848,Z 276.884,A -85,B 0,C 180,E1 -14408.449,E2 -14408.449} C_VEL
LIN {X 0,Y 336.246,Z 271.402,A -85,B 0,C 180,E1 -14410.234,E2 -14410.234} C_VEL
LIN {X 0,Y 337.687,Z 265.368,A -85,B 0,C 180,E1 -14411.708,E2 -14411.708} C_VEL
LIN {X 0,Y 339.31,Z 257.741,A -85,B 0,C 180,E1 -14413.17,E2 -14413.17} C_VEL
LIN {X 0,Y 340.902,Z 249.166,A -85,B 0,C 180,E1 -14414.476,E2 -14414.476} C_VEL
LIN {X 0,Y 340.306,Z 239.888,A -85,B 0,C 180,E1 -14415.837,E2 -14415.837} C_VEL
LIN {X 0,Y 338.454,Z 229.759,A -85,B 0,C 180,E1 -14417.213,E2 -14417.213} C_VEL
LIN {X 0,Y 335.129,Z 217.959,A -85,B 0,C 180,E1 -14418.748,E2 -14418.748} C_VEL
LIN {X 0,Y 335.971,Z 212.412,A -85,B 0,C 180,E1 -14422.119,E2 -14422.119} C_VEL
LIN {X 0,Y 337.206,Z 206.543,A -85,B 0,C 180,E1 -14425.956,E2 -14425.956} C_VEL
LIN {X 0,Y 338.622,Z 201.254,A -85,B 0,C 180,E1 -14429.875,E2 -14429.875} C_VEL
LIN {X 0,Y 339.202,Z 198.967,A -85,B 0,C 180,E1 -14431.842,E2 -14431.842} C_VEL
LIN {X 0,Y 339.347,Z 196.871,A -85,B 0,C 180,E1 -14434.062,E2 -14434.062} C_VEL
LIN {X 0,Y 339.175,Z 194.81,A -85,B 0,C 180,E1 -14436.935,E2 -14436.935} C_VEL
LIN {X 0,Y 339.05,Z 193.389,A -85,B 0,C 180,E1 -14439.985,E2 -14439.985} C_VEL
LIN {X 0,Y 339.078,Z 192.79,A -85,B 0,C 180,E1 -14443.156,E2 -14443.156} C_VEL
LIN {X 0,Y 339.278,Z 193.178,A -85,B 0,C 180,E1 -14446.47,E2 -14446.47} C_VEL
LIN {X 0,Y 339.49,Z 193.942,A -85,B 0,C 180,E1 -14448.511,E2 -14448.511} C_VEL
LIN {X 0,Y 339.923,Z 196.106,A -85,B 0,C 180,E1 -14451.782,E2 -14451.782} C_VEL
LIN {X 0,Y 340.474,Z 198.945,A -85,B 0,C 180,E1 -14454.69,E2 -14454.69} C_VEL
LIN {X 0,Y 341.208,Z 202.595,A -85,B 0,C 180,E1 -14457.618,E2 -14457.618} C_VEL
LIN {X 0,Y 341.619,Z 205.926,A -85,B 0,C 180,E1 -14459.775,E2 -14459.775} C_VEL
LIN {X 0,Y 341.169,Z 208.32,A -85,B 0,C 180,E1 -14461.045,E2 -14461.045} C_VEL
LIN {X 0,Y 338.964,Z 215.187,A -85,B 0,C 180,E1 -14464.187,E2 -14464.187} C_VEL
LIN {X 0,Y 337.685,Z 220.506,A -85,B 0,C 180,E1 -14466.407,E2 -14466.407} C_VEL
LIN {X 0,Y 341.008,Z 233.663,A -85,B 0,C 180,E1 -14467.586,E2 -14467.586} C_VEL
LIN {X 0,Y 342.418,Z 243.281,A -85,B 0,C 180,E1 -14468.483,E2 -14468.483} C_VEL
LIN {X 0,Y 342.675,Z 250.889,A -85,B 0,C 180,E1 -14469.216,E2 -14469.216} C_VEL
LIN {X 0,Y 341.725,Z 259.093,A -85,B 0,C 180,E1 -14470.005,E2 -14470.005} C_VEL
LIN {X 0,Y 339.833,Z 270.4,A -85,B 0,C 180,E1 -14471.302,E2 -14471.302} C_VEL
LIN {X 0,Y 337.962,Z 280.494,A -85,B 0,C 180,E1 -14472.761,E2 -14472.761} C_VEL
LIN {X 0,Y 336.372,Z 288.78,A -85,B 0,C 180,E1 -14474.238,E2 -14474.238} C_VEL
LIN {X 0,Y 335.064,Z 296.873,A -85,B 0,C 180,E1 -14476.04,E2 -14476.04} C_VEL
LIN {X 0,Y 333.727,Z 303.439,A -85,B 0,C 180,E1 -14477.841,E2 -14477.841} C_VEL
LIN {X 0,Y 332.96,Z 308.697,A -85,B 0,C 180,E1 -14479.663,E2 -14479.663} C_VEL
LIN {X 0,Y 332.44,Z 312.778,A -85,B 0,C 180,E1 -14481.488,E2 -14481.488} C_VEL
LIN {X 0,Y 332.195,Z 314.89,A -85,B 0,C 180,E1 -14482.706,E2 -14482.706} C_VEL
LIN {X 0,Y 332.093,Z 316.773,A -85,B 0,C 180,E1 -14484.072,E2 -14484.072} C_VEL
LIN {X 0,Y 332.041,Z 318.662,A -85,B 0,C 180,E1 -14486.358,E2 -14486.358} C_VEL
LIN {X 0,Y 332.057,Z 319.072,A -85,B 0,C 180,E1 -14487.572,E2 -14487.572} C_VEL
LIN {X 0,Y 332.256,Z 319.069,A -85,B 0,C 180,E1 -14488.786,E2 -14488.786} C_VEL
LIN {X 0,Y 332.273,Z 318.588,A -85,B 0,C 180,E1 -14489.998,E2 -14489.998} C_VEL
LIN {X 0,Y 332.301,Z 317.696,A -85,B 0,C 180,E1 -14491.21,E2 -14491.21} C_VEL
LIN {X 0,Y 332.298,Z 316.345,A -85,B 0,C 180,E1 -14492.422,E2 -14492.422} C_VEL
LIN {X 0,Y 332.188,Z 313.383,A -85,B 0,C 180,E1 -14494.245,E2 -14494.245} C_VEL
LIN {X 0,Y 332.312,Z 308.722,A -85,B 0,C 180,E1 -14496.28,E2 -14496.28} C_VEL
LIN {X 0,Y 332.451,Z 302.85,A -85,B 0,C 180,E1 -14498.202,E2 -14498.202} C_VEL
LIN {X 0,Y 332.723,Z 295.625,A -85,B 0,C 180,E1 -14500.034,E2 -14500.034} C_VEL
LIN {X 0,Y 333.137,Z 288.191,A -85,B 0,C 180,E1 -14501.559,E2 -14501.559} C_VEL
LIN {X 0,Y 333.666,Z 279.055,A -85,B 0,C 180,E1 -14503.085,E2 -14503.085} C_VEL
LIN {X 0,Y 334.309,Z 268.839,A -85,B 0,C 180,E1 -14504.454,E2 -14504.454} C_VEL
LIN {X 0,Y 335.132,Z 257.413,A -85,B 0,C 180,E1 -14505.67,E2 -14505.67} C_VEL
LIN {X 0,Y 335.686,Z 245.439,A -85,B 0,C 180,E1 -14506.65,E2 -14506.65} C_VEL
LIN {X 0,Y 334.492,Z 232.78,A -85,B 0,C 180,E1 -14507.439,E2 -14507.439} C_VEL
LIN {X 0,Y 333.665,Z 220.088,A -85,B 0,C 180,E1 -14508.019,E2 -14508.019} C_VEL
LIN {X 0,Y 334.866,Z 207.993,A -85,B 0,C 180,E1 -14512.194,E2 -14512.194} C_VEL
LIN {X 0,Y 336.313,Z 197.018,A -85,B 0,C 180,E1 -14516.027,E2 -14516.027} C_VEL
LIN {X 0,Y 337.204,Z 189.636,A -85,B 0,C 180,E1 -14518.641,E2 -14518.641} C_VEL
LIN {X 0,Y 336.088,Z 183.488,A -85,B 0,C 180,E1 -14520.978,E2 -14520.978} C_VEL
LIN {X 0,Y 333.938,Z 172.141,A -85,B 0,C 180,E1 -14525.442,E2 -14525.442} C_VEL
LIN {X 0,Y 333.7,Z 170.926,A -85,B 0,C 180,E1 -14525.967,E2 -14525.967} C_VEL
LIN {X 0,Y 333.639,Z 170.924,A -85,B 0,C 180,E1 -14529.19,E2 -14529.19} C_VEL
LIN {X 0,Y 333.626,Z 170.929,A -85,B 0,C 180,E1 -14532.498,E2 -14532.498} C_VEL
LIN {X 0,Y 333.66,Z 170.922,A -85,B 0,C 180,E1 -14535.965,E2 -14535.965} C_VEL
LIN {X 0,Y 333.692,Z 170.916,A -85,B 0,C 180,E1 -14539.303,E2 -14539.303} C_VEL
LIN {X 0,Y 333.656,Z 170.92,A -85,B 0,C 180,E1 -14543.166,E2 -14543.166} C_VEL
LIN {X 0,Y 333.625,Z 170.925,A -85,B 0,C 180,E1 -14546.79,E2 -14546.79} C_VEL
LIN {X 0,Y 333.691,Z 170.919,A -85,B 0,C 180,E1 -14549.709,E2 -14549.709} C_VEL
LIN {X 0,Y 333.732,Z 170.913,A -85,B 0,C 180,E1 -14552.4,E2 -14552.4} C_VEL
LIN {X 0,Y 333.713,Z 170.914,A -85,B 0,C 180,E1 -14555.089,E2 -14555.089} C_VEL
LIN {X 0,Y 333.662,Z 170.92,A -85,B 0,C 180,E1 -14559.018,E2 -14559.018} C_VEL
LIN {X 0,Y 333.781,Z 170.91,A -85,B 0,C 180,E1 -14561.589,E2 -14561.589} C_VEL
LIN {X 0,Y 333.794,Z 170.908,A -85,B 0,C 180,E1 -14565.576,E2 -14565.576} C_VEL
LIN {X 0,Y 333.822,Z 170.903,A -85,B 0,C 180,E1 -14569.078,E2 -14569.078} C_VEL
LIN {X 0,Y 334,Z 170.879,A -85,B 0,C 180,E1 -14572.747,E2 -14572.747} C_VEL
LIN {X 0,Y 333.801,Z 170.908,A -85,B 0,C 180,E1 -14575.169,E2 -14575.169} C_VEL
LIN {X 0,Y 334.118,Z 170.864,A -85,B 0,C 180,E1 -14577.589,E2 -14577.589} C_VEL
LIN {X 0,Y 334.232,Z 170.849,A -85,B 0,C 180,E1 -14580,E2 -14580} C_VEL
LIN {X 0,Y 334.088,Z 170.868,A -85,B 0,C 180,E1 -14582.411,E2 -14582.411} C_VEL
LIN {X 0,Y 334.011,Z 170.878,A -85,B 0,C 180,E1 -14587.253,E2 -14587.253} C_VEL
LIN {X 0,Y 333.823,Z 170.903,A -85,B 0,C 180,E1 -14590.922,E2 -14590.922} C_VEL
LIN {X 0,Y 333.794,Z 170.908,A -85,B 0,C 180,E1 -14594.635,E2 -14594.635} C_VEL
LIN {X 0,Y 333.784,Z 170.908,A -85,B 0,C 180,E1 -14598.657,E2 -14598.657} C_VEL
LIN {X 0,Y 333.68,Z 170.923,A -85,B 0,C 180,E1 -14602.279,E2 -14602.279} C_VEL
LIN {X 0,Y 333.689,Z 170.917,A -85,B 0,C 180,E1 -14605.096,E2 -14605.096} C_VEL
LIN {X 0,Y 333.642,Z 170.922,A -85,B 0,C 180,E1 -14608.979,E2 -14608.979} C_VEL
LIN {X 0,Y 333.631,Z 170.924,A -85,B 0,C 180,E1 -14612.588,E2 -14612.588} C_VEL
LIN {X 0,Y 333.666,Z 170.922,A -85,B 0,C 180,E1 -14616.14,E2 -14616.14} C_VEL
LIN {X 0,Y 333.637,Z 170.924,A -85,B 0,C 180,E1 -14619.194,E2 -14619.194} C_VEL
LIN {X 0,Y 333.623,Z 170.925,A -85,B 0,C 180,E1 -14622.502,E2 -14622.502} C_VEL
LIN {X 0,Y 333.613,Z 170.927,A -85,B 0,C 180,E1 -14625.961,E2 -14625.961} C_VEL
LIN {X 0,Y 333.639,Z 170.928,A -85,B 0,C 180,E1 -14629.317,E2 -14629.317} C_VEL
LIN {X 0,Y 333.657,Z 170.925,A -85,B 0,C 180,E1 -14633.17,E2 -14633.17} C_VEL
LIN {X 0,Y 333.667,Z 170.923,A -85,B 0,C 180,E1 -14635.343,E2 -14635.343} C_VEL
LIN {X 0,Y 333.697,Z 170.916,A -85,B 0,C 180,E1 -14639.712,E2 -14639.712} C_VEL
LIN {X 0,Y 333.739,Z 170.912,A -85,B 0,C 180,E1 -14642.403,E2 -14642.403} C_VEL
LIN {X 0,Y 333.722,Z 170.915,A -85,B 0,C 180,E1 -14645.093,E2 -14645.093} C_VEL
LIN {X 0,Y 333.682,Z 170.92,A -85,B 0,C 180,E1 -14649.022,E2 -14649.022} C_VEL
LIN {X 0,Y 333.791,Z 170.904,A -85,B 0,C 180,E1 -14651.592,E2 -14651.592} C_VEL
LIN {X 0,Y 333.806,Z 170.902,A -85,B 0,C 180,E1 -14655.579,E2 -14655.579} C_VEL
LIN {X 0,Y 333.833,Z 170.899,A -85,B 0,C 180,E1 -14659.08,E2 -14659.08} C_VEL
LIN {X 0,Y 334.026,Z 170.876,A -85,B 0,C 180,E1 -14662.75,E2 -14662.75} C_VEL
LIN {X 0,Y 333.811,Z 170.901,A -85,B 0,C 180,E1 -14665.171,E2 -14665.171} C_VEL
LIN {X 0,Y 334.107,Z 170.866,A -85,B 0,C 180,E1 -14667.591,E2 -14667.591} C_VEL
LIN {X 0,Y 334.061,Z 170.87,A -85,B 0,C 180,E1 -14671.207,E2 -14671.207} C_VEL
LIN {X 0,Y 334.103,Z 170.866,A -85,B 0,C 180,E1 -14672.413,E2 -14672.413} C_VEL
LIN {X 0,Y 334.029,Z 170.876,A -85,B 0,C 180,E1 -14677.254,E2 -14677.254} C_VEL
LIN {X 0,Y 333.837,Z 170.899,A -85,B 0,C 180,E1 -14680.924,E2 -14680.924} C_VEL
LIN {X 0,Y 333.812,Z 170.901,A -85,B 0,C 180,E1 -14684.636,E2 -14684.636} C_VEL
LIN {X 0,Y 333.8,Z 170.903,A -85,B 0,C 180,E1 -14688.656,E2 -14688.656} C_VEL
LIN {X 0,Y 333.653,Z 170.921,A -85,B 0,C 180,E1 -14692.283,E2 -14692.283} C_VEL
LIN {X 0,Y 333.662,Z 170.925,A -85,B 0,C 180,E1 -14695.08,E2 -14695.08} C_VEL
LIN {X 0,Y 333.657,Z 170.926,A -85,B 0,C 180,E1 -14698.979,E2 -14698.979} C_VEL
LIN {X 0,Y 333.649,Z 170.924,A -85,B 0,C 180,E1 -14702.588,E2 -14702.588} C_VEL
LIN {X 0,Y 333.68,Z 170.918,A -85,B 0,C 180,E1 -14706.14,E2 -14706.14} C_VEL
LIN {X 0,Y 333.625,Z 170.926,A -85,B 0,C 180,E1 -14709.197,E2 -14709.197} C_VEL
LIN {X 0,Y 333.634,Z 170.928,A -85,B 0,C 180,E1 -14712.5,E2 -14712.5} C_VEL
LIN {X 0,Y 333.602,Z 170.929,A -85,B 0,C 180,E1 -14715.956,E2 -14715.956} C_VEL
LIN {X 0,Y 333.649,Z 170.921,A -85,B 0,C 180,E1 -14719.317,E2 -14719.317} C_VEL
LIN {X 0,Y 333.669,Z 170.919,A -85,B 0,C 180,E1 -14723.169,E2 -14723.169} C_VEL
LIN {X 0,Y 333.819,Z 171.103,A -85,B 0,C 180,E1 -14725.724,E2 -14725.724} C_VEL
LIN {X 0,Y 334.792,Z 177.053,A -85,B 0,C 180,E1 -14728.922,E2 -14728.922} C_VEL
LIN {X 0,Y 334.594,Z 181.325,A -85,B 0,C 180,E1 -14731.112,E2 -14731.112} C_VEL
LIN {X 0,Y 333.995,Z 188.678,A -85,B 0,C 180,E1 -14734.801,E2 -14734.801} C_VEL
LIN {X 0,Y 333.494,Z 196.173,A -85,B 0,C 180,E1 -14738.499,E2 -14738.499} C_VEL
LIN {X 0,Y 333.397,Z 197.411,A -85,B 0,C 180,E1 -14739.103,E2 -14739.103} C_VEL
LIN {X 0,Y 332.602,Z 199.408,A -85,B 0,C 180,E1 -14740.05,E2 -14740.05} C_VEL
LIN {X 0,Y 329.54,Z 202.764,A -85,B 0,C 180,E1 -14741.576,E2 -14741.576} C_VEL
LIN {X 0,Y 326.975,Z 205.46,A -85,B 0,C 180,E1 -14742.811,E2 -14742.811} C_VEL
LIN {X 0,Y 325.849,Z 207.489,A -85,B 0,C 180,E1 -14743.774,E2 -14743.774} C_VEL
LIN {X 0,Y 325.741,Z 208.162,A -85,B 0,C 180,E1 -14744.102,E2 -14744.102} C_VEL
LIN {X 0,Y 325.464,Z 216.393,A -85,B 0,C 180,E1 -14748.044,E2 -14748.044} C_VEL
LIN {X 0,Y 326.226,Z 227.742,A -85,B 0,C 180,E1 -14748.82,E2 -14748.82} C_VEL
LIN {X 0,Y 327.011,Z 236.717,A -85,B 0,C 180,E1 -14749.631,E2 -14749.631} C_VEL
LIN {X 0,Y 326.438,Z 247.53,A -85,B 0,C 180,E1 -14750.864,E2 -14750.864} C_VEL
LIN {X 0,Y 326.014,Z 256.91,A -85,B 0,C 180,E1 -14752.257,E2 -14752.257} C_VEL
LIN {X 0,Y 325.65,Z 265.032,A -85,B 0,C 180,E1 -14753.805,E2 -14753.805} C_VEL
LIN {X 0,Y 325.443,Z 271.352,A -85,B 0,C 180,E1 -14755.355,E2 -14755.355} C_VEL
LIN {X 0,Y 325.171,Z 276.241,A -85,B 0,C 180,E1 -14756.903,E2 -14756.903} C_VEL
LIN {X 0,Y 325.044,Z 280.478,A -85,B 0,C 180,E1 -14758.761,E2 -14758.761} C_VEL
LIN {X 0,Y 325.097,Z 282.424,A -85,B 0,C 180,E1 -14760,E2 -14760} C_VEL
LIN {X 0,Y 325.244,Z 283.707,A -85,B 0,C 180,E1 -14761.238,E2 -14761.238} C_VEL
LIN {X 0,Y 325.496,Z 284.338,A -85,B 0,C 180,E1 -14762.475,E2 -14762.475} C_VEL
LIN {X 0,Y 325.845,Z 284.329,A -85,B 0,C 180,E1 -14763.71,E2 -14763.71} C_VEL
LIN {X 0,Y 326.4,Z 283.687,A -85,B 0,C 180,E1 -14764.941,E2 -14764.941} C_VEL
LIN {X 0,Y 326.634,Z 282.468,A -85,B 0,C 180,E1 -14766.176,E2 -14766.176} C_VEL
LIN {X 0,Y 327.654,Z 279.397,A -85,B 0,C 180,E1 -14768.014,E2 -14768.014} C_VEL
LIN {X 0,Y 328.406,Z 276.509,A -85,B 0,C 180,E1 -14769.236,E2 -14769.236} C_VEL
LIN {X 0,Y 329.968,Z 270.74,A -85,B 0,C 180,E1 -14771.052,E2 -14771.052} C_VEL
LIN {X 0,Y 331.554,Z 264.462,A -85,B 0,C 180,E1 -14772.549,E2 -14772.549} C_VEL
LIN {X 0,Y 333.361,Z 256.526,A -85,B 0,C 180,E1 -14774.031,E2 -14774.031} C_VEL
LIN {X 0,Y 334.513,Z 250.146,A -85,B 0,C 180,E1 -14775.022,E2 -14775.022} C_VEL
LIN {X 0,Y 333.922,Z 240.727,A -85,B 0,C 180,E1 -14776.48,E2 -14776.48} C_VEL
LIN {X 0,Y 332.236,Z 231.393,A -85,B 0,C 180,E1 -14777.837,E2 -14777.837} C_VEL
LIN {X 0,Y 329.475,Z 221.534,A -85,B 0,C 180,E1 -14779.222,E2 -14779.222} C_VEL
LIN {X 0,Y 328.454,Z 218.093,A -85,B 0,C 180,E1 -14779.695,E2 -14779.695} C_VEL
LIN {X 0,Y 329.633,Z 211.566,A -85,B 0,C 180,E1 -14783.897,E2 -14783.897} C_VEL
LIN {X 0,Y 330.635,Z 207.459,A -85,B 0,C 180,E1 -14786.776,E2 -14786.776} C_VEL
LIN {X 0,Y 331.758,Z 203.65,A -85,B 0,C 180,E1 -14789.707,E2 -14789.707} C_VEL
LIN {X 0,Y 332.502,Z 200.777,A -85,B 0,C 180,E1 -14792.275,E2 -14792.275} C_VEL
LIN {X 0,Y 332.579,Z 198.646,A -85,B 0,C 180,E1 -14794.789,E2 -14794.789} C_VEL
LIN {X 0,Y 332.482,Z 196.788,A -85,B 0,C 180,E1 -14797.807,E2 -14797.807} C_VEL
LIN {X 0,Y 332.406,Z 195.673,A -85,B 0,C 180,E1 -14800.952,E2 -14800.952} C_VEL
LIN {X 0,Y 332.494,Z 195.412,A -85,B 0,C 180,E1 -14804.229,E2 -14804.229} C_VEL
LIN {X 0,Y 332.763,Z 196.127,A -85,B 0,C 180,E1 -14807.478,E2 -14807.478} C_VEL
LIN {X 0,Y 333.13,Z 197.887,A -85,B 0,C 180,E1 -14810.733,E2 -14810.733} C_VEL
LIN {X 0,Y 333.655,Z 200.546,A -85,B 0,C 180,E1 -14813.857,E2 -14813.857} C_VEL
LIN {X 0,Y 334.412,Z 204.467,A -85,B 0,C 180,E1 -14817.208,E2 -14817.208} C_VEL
LIN {X 0,Y 334.866,Z 208.204,A -85,B 0,C 180,E1 -14819.753,E2 -14819.753} C_VEL
LIN {X 0,Y 334.253,Z 210.726,A -85,B 0,C 180,E1 -14821.078,E2 -14821.078} C_VEL
LIN {X 0,Y 331.981,Z 217.552,A -85,B 0,C 180,E1 -14824.278,E2 -14824.278} C_VEL
LIN {X 0,Y 331.23,Z 220.349,A -85,B 0,C 180,E1 -14825.513,E2 -14825.513} C_VEL
LIN {X 0,Y 334.634,Z 233.602,A -85,B 0,C 180,E1 -14826.808,E2 -14826.808} C_VEL
LIN {X 0,Y 336.205,Z 244.432,A -85,B 0,C 180,E1 -14827.895,E2 -14827.895} C_VEL
LIN {X 0,Y 336.335,Z 253.627,A -85,B 0,C 180,E1 -14828.836,E2 -14828.836} C_VEL
LIN {X 0,Y 334.546,Z 264.951,A -85,B 0,C 180,E1 -14830.038,E2 -14830.038} C_VEL
LIN {X 0,Y 332.424,Z 275.961,A -85,B 0,C 180,E1 -14831.509,E2 -14831.509} C_VEL
LIN {X 0,Y 330.562,Z 284.909,A -85,B 0,C 180,E1 -14832.994,E2 -14832.994} C_VEL
LIN {X 0,Y 329.092,Z 292.352,A -85,B 0,C 180,E1 -14834.516,E2 -14834.516} C_VEL
LIN {X 0,Y 327.711,Z 299.642,A -85,B 0,C 180,E1 -14836.353,E2 -14836.353} C_VEL
LIN {X 0,Y 326.493,Z 305.561,A -85,B 0,C 180,E1 -14838.198,E2 -14838.198} C_VEL
LIN {X 0,Y 325.739,Z 310.245,A -85,B 0,C 180,E1 -14840.059,E2 -14840.059} C_VEL
LIN {X 0,Y 325.247,Z 313.83,A -85,B 0,C 180,E1 -14841.924,E2 -14841.924} C_VEL
LIN {X 0,Y 325.001,Z 316.724,A -85,B 0,C 180,E1 -14844.117,E2 -14844.117} C_VEL
LIN {X 0,Y 324.965,Z 318.305,A -85,B 0,C 180,E1 -14846.278,E2 -14846.278} C_VEL
LIN {X 0,Y 324.967,Z 318.65,A -85,B 0,C 180,E1 -14847.519,E2 -14847.519} C_VEL
LIN {X 0,Y 325.192,Z 318.541,A -85,B 0,C 180,E1 -14848.76,E2 -14848.76} C_VEL
LIN {X 0,Y 325.214,Z 318.006,A -85,B 0,C 180,E1 -14849.998,E2 -14849.998} C_VEL
LIN {X 0,Y 325.243,Z 317.045,A -85,B 0,C 180,E1 -14851.236,E2 -14851.236} C_VEL
LIN {X 0,Y 325.222,Z 315.579,A -85,B 0,C 180,E1 -14852.475,E2 -14852.475} C_VEL
LIN {X 0,Y 325.132,Z 312.492,A -85,B 0,C 180,E1 -14854.337,E2 -14854.337} C_VEL
LIN {X 0,Y 325.248,Z 308.019,A -85,B 0,C 180,E1 -14856.292,E2 -14856.292} C_VEL
LIN {X 0,Y 325.391,Z 301.593,A -85,B 0,C 180,E1 -14858.381,E2 -14858.381} C_VEL
LIN {X 0,Y 325.667,Z 294.192,A -85,B 0,C 180,E1 -14860.253,E2 -14860.253} C_VEL
LIN {X 0,Y 326.15,Z 286.533,A -85,B 0,C 180,E1 -14861.81,E2 -14861.81} C_VEL
LIN {X 0,Y 326.758,Z 277.071,A -85,B 0,C 180,E1 -14863.366,E2 -14863.366} C_VEL
LIN {X 0,Y 327.295,Z 267.767,A -85,B 0,C 180,E1 -14864.612,E2 -14864.612} C_VEL
LIN {X 0,Y 328.112,Z 256.499,A -85,B 0,C 180,E1 -14865.815,E2 -14865.815} C_VEL
LIN {X 0,Y 328.61,Z 245.946,A -85,B 0,C 180,E1 -14866.699,E2 -14866.699} C_VEL
LIN {X 0,Y 327.439,Z 233.293,A -85,B 0,C 180,E1 -14867.525,E2 -14867.525} C_VEL
LIN {X 0,Y 326.593,Z 220.076,A -85,B 0,C 180,E1 -14868.139,E2 -14868.139} C_VEL
LIN {X 0,Y 327.974,Z 207.275,A -85,B 0,C 180,E1 -14872.686,E2 -14872.686} C_VEL
LIN {X 0,Y 329.442,Z 196.335,A -85,B 0,C 180,E1 -14876.612,E2 -14876.612} C_VEL
LIN {X 0,Y 330.159,Z 191.025,A -85,B 0,C 180,E1 -14878.538,E2 -14878.538} C_VEL
LIN {X 0,Y 329.174,Z 185.082,A -85,B 0,C 180,E1 -14880.822,E2 -14880.822} C_VEL
LIN {X 0,Y 327.077,Z 174.047,A -85,B 0,C 180,E1 -14885.262,E2 -14885.262} C_VEL
LIN {X 0,Y 326.652,Z 171.801,A -85,B 0,C 180,E1 -14886.273,E2 -14886.273} C_VEL
LIN {X 0,Y 326.583,Z 171.803,A -85,B 0,C 180,E1 -14890.207,E2 -14890.207} C_VEL
LIN {X 0,Y 326.576,Z 171.802,A -85,B 0,C 180,E1 -14893.52,E2 -14893.52} C_VEL
LIN {X 0,Y 326.619,Z 171.798,A -85,B 0,C 180,E1 -14897.016,E2 -14897.016} C_VEL
LIN {X 0,Y 326.634,Z 171.797,A -85,B 0,C 180,E1 -14900.764,E2 -14900.764} C_VEL
LIN {X 0,Y 326.602,Z 171.802,A -85,B 0,C 180,E1 -14904.479,E2 -14904.479} C_VEL
LIN {X 0,Y 326.596,Z 171.801,A -85,B 0,C 180,E1 -14907.454,E2 -14907.454} C_VEL
LIN {X 0,Y 326.649,Z 171.796,A -85,B 0,C 180,E1 -14910.34,E2 -14910.34} C_VEL
LIN {X 0,Y 326.673,Z 171.791,A -85,B 0,C 180,E1 -14913.141,E2 -14913.141} C_VEL
LIN {X 0,Y 326.636,Z 171.8,A -85,B 0,C 180,E1 -14915.87,E2 -14915.87} C_VEL
LIN {X 0,Y 326.647,Z 171.797,A -85,B 0,C 180,E1 -14919.864,E2 -14919.864} C_VEL
LIN {X 0,Y 326.686,Z 171.789,A -85,B 0,C 180,E1 -14922.471,E2 -14922.471} C_VEL
LIN {X 0,Y 326.746,Z 171.781,A -85,B 0,C 180,E1 -14926.314,E2 -14926.314} C_VEL
LIN {X 0,Y 326.799,Z 171.775,A -85,B 0,C 180,E1 -14930.093,E2 -14930.093} C_VEL
LIN {X 0,Y 326.954,Z 171.756,A -85,B 0,C 180,E1 -14932.59,E2 -14932.59} C_VEL
LIN {X 0,Y 326.768,Z 171.783,A -85,B 0,C 180,E1 -14935.065,E2 -14935.065} C_VEL
LIN {X 0,Y 327.055,Z 171.744,A -85,B 0,C 180,E1 -14937.537,E2 -14937.537} C_VEL
LIN {X 0,Y 327.183,Z 171.727,A -85,B 0,C 180,E1 -14940,E2 -14940} C_VEL
LIN {X 0,Y 327.029,Z 171.748,A -85,B 0,C 180,E1 -14942.463,E2 -14942.463} C_VEL
LIN {X 0,Y 326.955,Z 171.754,A -85,B 0,C 180,E1 -14946.692,E2 -14946.692} C_VEL
LIN {X 0,Y 326.801,Z 171.775,A -85,B 0,C 180,E1 -14949.907,E2 -14949.907} C_VEL
LIN {X 0,Y 326.746,Z 171.781,A -85,B 0,C 180,E1 -14953.686,E2 -14953.686} C_VEL
LIN {X 0,Y 326.686,Z 171.789,A -85,B 0,C 180,E1 -14957.529,E2 -14957.529} C_VEL
LIN {X 0,Y 326.661,Z 171.796,A -85,B 0,C 180,E1 -14960.135,E2 -14960.135} C_VEL
LIN {X 0,Y 326.633,Z 171.8,A -85,B 0,C 180,E1 -14964.13,E2 -14964.13} C_VEL
LIN {X 0,Y 326.609,Z 171.802,A -85,B 0,C 180,E1 -14968.255,E2 -14968.255} C_VEL
LIN {X 0,Y 326.561,Z 171.804,A -85,B 0,C 180,E1 -14971.098,E2 -14971.098} C_VEL
LIN {X 0,Y 326.595,Z 171.804,A -85,B 0,C 180,E1 -14974.021,E2 -14974.021} C_VEL
LIN {X 0,Y 326.618,Z 171.798,A -85,B 0,C 180,E1 -14977.241,E2 -14977.241} C_VEL
LIN {X 0,Y 326.568,Z 171.805,A -85,B 0,C 180,E1 -14981.133,E2 -14981.133} C_VEL
LIN {X 0,Y 326.546,Z 171.806,A -85,B 0,C 180,E1 -14984.75,E2 -14984.75} C_VEL
LIN {X 0,Y 326.568,Z 171.804,A -85,B 0,C 180,E1 -14988.156,E2 -14988.156} C_VEL
LIN {X 0,Y 326.615,Z 171.802,A -85,B 0,C 180,E1 -14991.393,E2 -14991.393} C_VEL
LIN {X 0,Y 326.612,Z 171.801,A -85,B 0,C 180,E1 -14994.853,E2 -14994.853} C_VEL
LIN {X 0,Y 326.601,Z 171.801,A -85,B 0,C 180,E1 -14997.458,E2 -14997.458} C_VEL
LIN {X 0,Y 326.655,Z 171.793,A -85,B 0,C 180,E1 -15000.343,E2 -15000.343} C_VEL
LIN {X 0,Y 326.685,Z 171.791,A -85,B 0,C 180,E1 -15004.518,E2 -15004.518} C_VEL
LIN {X 0,Y 326.645,Z 171.798,A -85,B 0,C 180,E1 -15008.548,E2 -15008.548} C_VEL
LIN {X 0,Y 326.741,Z 171.783,A -85,B 0,C 180,E1 -15011.18,E2 -15011.18} C_VEL
LIN {X 0,Y 326.761,Z 171.779,A -85,B 0,C 180,E1 -15015.435,E2 -15015.435} C_VEL
LIN {X 0,Y 326.769,Z 171.78,A -85,B 0,C 180,E1 -15018.841,E2 -15018.841} C_VEL
LIN {X 0,Y 326.98,Z 171.755,A -85,B 0,C 180,E1 -15022.592,E2 -15022.592} C_VEL
LIN {X 0,Y 326.778,Z 171.777,A -85,B 0,C 180,E1 -15025.067,E2 -15025.067} C_VEL
LIN {X 0,Y 327.047,Z 171.745,A -85,B 0,C 180,E1 -15027.539,E2 -15027.539} C_VEL
LIN {X 0,Y 327.032,Z 171.746,A -85,B 0,C 180,E1 -15031.233,E2 -15031.233} C_VEL
LIN {X 0,Y 327.044,Z 171.745,A -85,B 0,C 180,E1 -15032.465,E2 -15032.465} C_VEL
LIN {X 0,Y 326.999,Z 171.752,A -85,B 0,C 180,E1 -15036.171,E2 -15036.171} C_VEL
LIN {X 0,Y 326.918,Z 171.76,A -85,B 0,C 180,E1 -15038.657,E2 -15038.657} C_VEL
LIN {X 0,Y 326.738,Z 171.782,A -85,B 0,C 180,E1 -15042.423,E2 -15042.423} C_VEL
LIN {X 0,Y 326.758,Z 171.781,A -85,B 0,C 180,E1 -15044.959,E2 -15044.959} C_VEL
LIN {X 0,Y 326.737,Z 171.784,A -85,B 0,C 180,E1 -15048.84,E2 -15048.84} C_VEL
LIN {X 0,Y 326.595,Z 171.802,A -85,B 0,C 180,E1 -15052.791,E2 -15052.791} C_VEL
LIN {X 0,Y 326.601,Z 171.803,A -85,B 0,C 180,E1 -15056.867,E2 -15056.867} C_VEL
LIN {X 0,Y 326.616,Z 171.8,A -85,B 0,C 180,E1 -15060.604,E2 -15060.604} C_VEL
LIN {X 0,Y 326.612,Z 171.798,A -85,B 0,C 180,E1 -15064.021,E2 -15064.021} C_VEL
LIN {X 0,Y 326.628,Z 171.797,A -85,B 0,C 180,E1 -15067.238,E2 -15067.238} C_VEL
LIN {X 0,Y 326.549,Z 171.807,A -85,B 0,C 180,E1 -15071.125,E2 -15071.125} C_VEL
LIN {X 0,Y 326.566,Z 171.804,A -85,B 0,C 180,E1 -15073.527,E2 -15073.527} C_VEL
LIN {X 0,Y 326.581,Z 171.803,A -85,B 0,C 180,E1 -15077.029,E2 -15077.029} C_VEL
LIN {X 0,Y 326.605,Z 171.8,A -85,B 0,C 180,E1 -15080.776,E2 -15080.776} C_VEL
LIN {X 0,Y 326.686,Z 171.79,A -85,B 0,C 180,E1 -15084.837,E2 -15084.837} C_VEL
LIN {X 0,Y 326.775,Z 172.01,A -85,B 0,C 180,E1 -15085.628,E2 -15085.628} C_VEL
LIN {X 0,Y 327.775,Z 178.287,A -85,B 0,C 180,E1 -15089.057,E2 -15089.057} C_VEL
LIN {X 0,Y 327.434,Z 183.629,A -85,B 0,C 180,E1 -15091.822,E2 -15091.822} C_VEL
LIN {X 0,Y 326.854,Z 190.29,A -85,B 0,C 180,E1 -15095.21,E2 -15095.21} C_VEL
LIN {X 0,Y 326.322,Z 198.195,A -85,B 0,C 180,E1 -15099.185,E2 -15099.185} C_VEL
LIN {X 0,Y 325.935,Z 204.755,A -85,B 0,C 180,E1 -15102.43,E2 -15102.43} C_VEL
LIN {X 0,Y 325.741,Z 208.162,A -85,B 0,C 180,E1 -15104.102,E2 -15104.102} C_VEL
LIN {X 0,Y 325.012,Z 209.521,A -85,B 0,C 180,E1 -15104.746,E2 -15104.746} C_VEL
LIN {X 0,Y 322.067,Z 211.708,A -85,B 0,C 180,E1 -15105.746,E2 -15105.746} C_VEL
LIN {X 0,Y 319.112,Z 213.901,A -85,B 0,C 180,E1 -15106.763,E2 -15106.763} C_VEL
LIN {X 0,Y 318.394,Z 215.27,A -85,B 0,C 180,E1 -15107.426,E2 -15107.426} C_VEL
LIN {X 0,Y 318.374,Z 216.332,A -85,B 0,C 180,E1 -15107.935,E2 -15107.935} C_VEL
LIN {X 0,Y 319.129,Z 227.693,A -85,B 0,C 180,E1 -15108.729,E2 -15108.729} C_VEL
LIN {X 0,Y 319.935,Z 236.71,A -85,B 0,C 180,E1 -15109.559,E2 -15109.559} C_VEL
LIN {X 0,Y 319.348,Z 247.545,A -85,B 0,C 180,E1 -15110.819,E2 -15110.819} C_VEL
LIN {X 0,Y 318.981,Z 256.042,A -85,B 0,C 180,E1 -15112.085,E2 -15112.085} C_VEL
LIN {X 0,Y 318.57,Z 264.423,A -85,B 0,C 180,E1 -15113.667,E2 -15113.667} C_VEL
LIN {X 0,Y 318.382,Z 270.973,A -85,B 0,C 180,E1 -15115.252,E2 -15115.252} C_VEL
LIN {X 0,Y 318.092,Z 276.024,A -85,B 0,C 180,E1 -15116.834,E2 -15116.834} C_VEL
LIN {X 0,Y 317.949,Z 280.474,A -85,B 0,C 180,E1 -15118.734,E2 -15118.734} C_VEL
LIN {X 0,Y 317.998,Z 282.542,A -85,B 0,C 180,E1 -15120,E2 -15120} C_VEL
LIN {X 0,Y 318.151,Z 283.95,A -85,B 0,C 180,E1 -15121.266,E2 -15121.266} C_VEL
LIN {X 0,Y 318.414,Z 284.723,A -85,B 0,C 180,E1 -15122.53,E2 -15122.53} C_VEL
LIN {X 0,Y 318.807,Z 284.864,A -85,B 0,C 180,E1 -15123.792,E2 -15123.792} C_VEL
LIN {X 0,Y 319.358,Z 284.379,A -85,B 0,C 180,E1 -15125.05,E2 -15125.05} C_VEL
LIN {X 0,Y 319.639,Z 283.3,A -85,B 0,C 180,E1 -15126.312,E2 -15126.312} C_VEL
LIN {X 0,Y 320.72,Z 280.458,A -85,B 0,C 180,E1 -15128.189,E2 -15128.189} C_VEL
LIN {X 0,Y 322.039,Z 276.121,A -85,B 0,C 180,E1 -15130.055,E2 -15130.055} C_VEL
LIN {X 0,Y 323.454,Z 271.314,A -85,B 0,C 180,E1 -15131.572,E2 -15131.572} C_VEL
LIN {X 0,Y 325.188,Z 265.004,A -85,B 0,C 180,E1 -15133.116,E2 -15133.116} C_VEL
LIN {X 0,Y 327.124,Z 257.157,A -85,B 0,C 180,E1 -15134.622,E2 -15134.622} C_VEL
LIN {X 0,Y 328.131,Z 252.042,A -85,B 0,C 180,E1 -15135.454,E2 -15135.454} C_VEL
LIN {X 0,Y 327.708,Z 242.595,A -85,B 0,C 180,E1 -15137.013,E2 -15137.013} C_VEL
LIN {X 0,Y 326.075,Z 233.108,A -85,B 0,C 180,E1 -15138.492,E2 -15138.492} C_VEL
LIN {X 0,Y 323.388,Z 223.246,A -85,B 0,C 180,E1 -15139.987,E2 -15139.987} C_VEL
LIN {X 0,Y 321.813,Z 218.232,A -85,B 0,C 180,E1 -15140.744,E2 -15140.744} C_VEL
LIN {X 0,Y 322.928,Z 212.764,A -85,B 0,C 180,E1 -15144.425,E2 -15144.425} C_VEL
LIN {X 0,Y 324.431,Z 207.386,A -85,B 0,C 180,E1 -15148.462,E2 -15148.462} C_VEL
LIN {X 0,Y 325.445,Z 204.184,A -85,B 0,C 180,E1 -15151.217,E2 -15151.217} C_VEL
LIN {X 0,Y 325.791,Z 202.701,A -85,B 0,C 180,E1 -15152.719,E2 -15152.719} C_VEL
LIN {X 0,Y 325.845,Z 200.475,A -85,B 0,C 180,E1 -15155.616,E2 -15155.616} C_VEL
LIN {X 0,Y 325.797,Z 198.872,A -85,B 0,C 180,E1 -15158.725,E2 -15158.725} C_VEL
LIN {X 0,Y 325.793,Z 198.034,A -85,B 0,C 180,E1 -15161.969,E2 -15161.969} C_VEL
LIN {X 0,Y 325.951,Z 198.127,A -85,B 0,C 180,E1 -15165.36,E2 -15165.36} C_VEL
LIN {X 0,Y 326.306,Z 199.358,A -85,B 0,C 180,E1 -15168.924,E2 -15168.924} C_VEL
LIN {X 0,Y 326.6,Z 200.942,A -85,B 0,C 180,E1 -15171.386,E2 -15171.386} C_VEL
LIN {X 0,Y 327.198,Z 203.945,A -85,B 0,C 180,E1 -15174.708,E2 -15174.708} C_VEL
LIN {X 0,Y 327.81,Z 207.397,A -85,B 0,C 180,E1 -15177.588,E2 -15177.588} C_VEL
LIN {X 0,Y 328.08,Z 210.619,A -85,B 0,C 180,E1 -15179.773,E2 -15179.773} C_VEL
LIN {X 0,Y 326.802,Z 214.597,A -85,B 0,C 180,E1 -15181.851,E2 -15181.851} C_VEL
LIN {X 0,Y 324.877,Z 220.329,A -85,B 0,C 180,E1 -15184.555,E2 -15184.555} C_VEL
LIN {X 0,Y 327.992,Z 232.009,A -85,B 0,C 180,E1 -15185.806,E2 -15185.806} C_VEL
LIN {X 0,Y 329.953,Z 243.825,A -85,B 0,C 180,E1 -15187.081,E2 -15187.081} C_VEL
LIN {X 0,Y 330.293,Z 252.836,A -85,B 0,C 180,E1 -15188.066,E2 -15188.066} C_VEL
LIN {X 0,Y 329.216,Z 260.54,A -85,B 0,C 180,E1 -15188.883,E2 -15188.883} C_VEL
LIN {X 0,Y 326.869,Z 272.302,A -85,B 0,C 180,E1 -15190.368,E2 -15190.368} C_VEL
LIN {X 0,Y 325.004,Z 280.949,A -85,B 0,C 180,E1 -15191.725,E2 -15191.725} C_VEL
LIN {X 0,Y 322.837,Z 290.337,A -85,B 0,C 180,E1 -15193.559,E2 -15193.559} C_VEL
LIN {X 0,Y 321.348,Z 297.928,A -85,B 0,C 180,E1 -15195.431,E2 -15195.431} C_VEL
LIN {X 0,Y 319.861,Z 304.05,A -85,B 0,C 180,E1 -15197.306,E2 -15197.306} C_VEL
LIN {X 0,Y 318.956,Z 308.927,A -85,B 0,C 180,E1 -15199.203,E2 -15199.203} C_VEL
LIN {X 0,Y 318.343,Z 312.707,A -85,B 0,C 180,E1 -15201.108,E2 -15201.108} C_VEL
LIN {X 0,Y 318.069,Z 314.676,A -85,B 0,C 180,E1 -15202.38,E2 -15202.38} C_VEL
LIN {X 0,Y 317.902,Z 316.68,A -85,B 0,C 180,E1 -15204.176,E2 -15204.176} C_VEL
LIN {X 0,Y 317.89,Z 317.95,A -85,B 0,C 180,E1 -15206.195,E2 -15206.195} C_VEL
LIN {X 0,Y 317.88,Z 318.177,A -85,B 0,C 180,E1 -15207.464,E2 -15207.464} C_VEL
LIN {X 0,Y 318.128,Z 318.006,A -85,B 0,C 180,E1 -15208.732,E2 -15208.732} C_VEL
LIN {X 0,Y 318.157,Z 317.409,A -85,B 0,C 180,E1 -15209.998,E2 -15209.998} C_VEL
LIN {X 0,Y 318.187,Z 316.326,A -85,B 0,C 180,E1 -15211.264,E2 -15211.264} C_VEL
LIN {X 0,Y 318.073,Z 313.837,A -85,B 0,C 180,E1 -15213.165,E2 -15213.165} C_VEL
LIN {X 0,Y 318.161,Z 310.245,A -85,B 0,C 180,E1 -15215.067,E2 -15215.067} C_VEL
LIN {X 0,Y 318.193,Z 305.409,A -85,B 0,C 180,E1 -15216.975,E2 -15216.975} C_VEL
LIN {X 0,Y 318.375,Z 299.153,A -85,B 0,C 180,E1 -15218.887,E2 -15218.887} C_VEL
LIN {X 0,Y 318.723,Z 291.167,A -85,B 0,C 180,E1 -15220.801,E2 -15220.801} C_VEL
LIN {X 0,Y 319.227,Z 282.931,A -85,B 0,C 180,E1 -15222.393,E2 -15222.393} C_VEL
LIN {X 0,Y 319.928,Z 272.665,A -85,B 0,C 180,E1 -15223.981,E2 -15223.981} C_VEL
LIN {X 0,Y 320.618,Z 261.881,A -85,B 0,C 180,E1 -15225.314,E2 -15225.314} C_VEL
LIN {X 0,Y 321.382,Z 250.362,A -85,B 0,C 180,E1 -15226.424,E2 -15226.424} C_VEL
LIN {X 0,Y 321.386,Z 244.115,A -85,B 0,C 180,E1 -15226.922,E2 -15226.922} C_VEL
LIN {X 0,Y 320.175,Z 231.413,A -85,B 0,C 180,E1 -15227.73,E2 -15227.73} C_VEL
LIN {X 0,Y 319.525,Z 220.168,A -85,B 0,C 180,E1 -15228.234,E2 -15228.234} C_VEL
LIN {X 0,Y 320.797,Z 208.416,A -85,B 0,C 180,E1 -15232.514,E2 -15232.514} C_VEL
LIN {X 0,Y 322.4,Z 197.147,A -85,B 0,C 180,E1 -15236.65,E2 -15236.65} C_VEL
LIN {X 0,Y 323.119,Z 191.955,A -85,B 0,C 180,E1 -15238.586,E2 -15238.586} C_VEL
LIN {X 0,Y 322.175,Z 186.285,A -85,B 0,C 180,E1 -15240.827,E2 -15240.827} C_VEL
LIN {X 0,Y 320.154,Z 175.591,A -85,B 0,C 180,E1 -15245.206,E2 -15245.206} C_VEL
LIN {X 0,Y 319.602,Z 172.678,A -85,B 0,C 180,E1 -15246.517,E2 -15246.517} C_VEL
LIN {X 0,Y 319.551,Z 172.677,A -85,B 0,C 180,E1 -15249.667,E2 -15249.667} C_VEL
LIN {X 0,Y 319.555,Z 172.677,A -85,B 0,C 180,E1 -15253.467,E2 -15253.467} C_VEL
LIN {X 0,Y 319.594,Z 172.673,A -85,B 0,C 180,E1 -15257.023,E2 -15257.023} C_VEL
LIN {X 0,Y 319.575,Z 172.68,A -85,B 0,C 180,E1 -15260.375,E2 -15260.375} C_VEL
LIN {X 0,Y 319.549,Z 172.678,A -85,B 0,C 180,E1 -15263.571,E2 -15263.571} C_VEL
LIN {X 0,Y 319.566,Z 172.677,A -85,B 0,C 180,E1 -15266.685,E2 -15266.685} C_VEL
LIN {X 0,Y 319.58,Z 172.676,A -85,B 0,C 180,E1 -15269.615,E2 -15269.615} C_VEL
LIN {X 0,Y 319.605,Z 172.672,A -85,B 0,C 180,E1 -15272.498,E2 -15272.498} C_VEL
LIN {X 0,Y 319.59,Z 172.674,A -85,B 0,C 180,E1 -15275.303,E2 -15275.303} C_VEL
LIN {X 0,Y 319.59,Z 172.675,A -85,B 0,C 180,E1 -15279.399,E2 -15279.399} C_VEL
LIN {X 0,Y 319.645,Z 172.667,A -85,B 0,C 180,E1 -15282.072,E2 -15282.072} C_VEL
LIN {X 0,Y 319.719,Z 172.658,A -85,B 0,C 180,E1 -15286.007,E2 -15286.007} C_VEL
LIN {X 0,Y 319.744,Z 172.655,A -85,B 0,C 180,E1 -15289.872,E2 -15289.872} C_VEL
LIN {X 0,Y 319.912,Z 172.632,A -85,B 0,C 180,E1 -15292.426,E2 -15292.426} C_VEL
LIN {X 0,Y 319.737,Z 172.658,A -85,B 0,C 180,E1 -15294.956,E2 -15294.956} C_VEL
LIN {X 0,Y 319.996,Z 172.624,A -85,B 0,C 180,E1 -15297.482,E2 -15297.482} C_VEL
LIN {X 0,Y 320.135,Z 172.604,A -85,B 0,C 180,E1 -15300,E2 -15300} C_VEL
LIN {X 0,Y 319.973,Z 172.627,A -85,B 0,C 180,E1 -15302.518,E2 -15302.518} C_VEL
LIN {X 0,Y 319.915,Z 172.631,A -85,B 0,C 180,E1 -15306.683,E2 -15306.683} C_VEL
LIN {X 0,Y 319.746,Z 172.654,A -85,B 0,C 180,E1 -15310.127,E2 -15310.127} C_VEL
LIN {X 0,Y 319.717,Z 172.66,A -85,B 0,C 180,E1 -15314.725,E2 -15314.725} C_VEL
LIN {X 0,Y 319.677,Z 172.662,A -85,B 0,C 180,E1 -15319.04,E2 -15319.04} C_VEL
LIN {X 0,Y 319.555,Z 172.677,A -85,B 0,C 180,E1 -15323.321,E2 -15323.321} C_VEL
LIN {X 0,Y 319.562,Z 172.681,A -85,B 0,C 180,E1 -15326.094,E2 -15326.094} C_VEL
LIN {X 0,Y 319.54,Z 172.679,A -85,B 0,C 180,E1 -15328.939,E2 -15328.939} C_VEL
LIN {X 0,Y 319.511,Z 172.687,A -85,B 0,C 180,E1 -15331.864,E2 -15331.864} C_VEL
LIN {X 0,Y 319.569,Z 172.678,A -85,B 0,C 180,E1 -15335.545,E2 -15335.545} C_VEL
LIN {X 0,Y 319.563,Z 172.679,A -85,B 0,C 180,E1 -15338.009,E2 -15338.009} C_VEL
LIN {X 0,Y 319.541,Z 172.684,A -85,B 0,C 180,E1 -15341.604,E2 -15341.604} C_VEL
LIN {X 0,Y 319.506,Z 172.686,A -85,B 0,C 180,E1 -15345.264,E2 -15345.264} C_VEL
LIN {X 0,Y 319.52,Z 172.682,A -85,B 0,C 180,E1 -15348.714,E2 -15348.714} C_VEL
LIN {X 0,Y 319.553,Z 172.677,A -85,B 0,C 180,E1 -15352.35,E2 -15352.35} C_VEL
LIN {X 0,Y 319.553,Z 172.682,A -85,B 0,C 180,E1 -15355.125,E2 -15355.125} C_VEL
LIN {X 0,Y 319.564,Z 172.681,A -85,B 0,C 180,E1 -15359.06,E2 -15359.06} C_VEL
LIN {X 0,Y 319.604,Z 172.673,A -85,B 0,C 180,E1 -15362.5,E2 -15362.5} C_VEL
LIN {X 0,Y 319.6,Z 172.673,A -85,B 0,C 180,E1 -15365.306,E2 -15365.306} C_VEL
LIN {X 0,Y 319.594,Z 172.673,A -85,B 0,C 180,E1 -15368.05,E2 -15368.05} C_VEL
LIN {X 0,Y 319.686,Z 172.663,A -85,B 0,C 180,E1 -15370.964,E2 -15370.964} C_VEL
LIN {X 0,Y 319.729,Z 172.655,A -85,B 0,C 180,E1 -15375.278,E2 -15375.278} C_VEL
LIN {X 0,Y 319.757,Z 172.653,A -85,B 0,C 180,E1 -15379.875,E2 -15379.875} C_VEL
LIN {X 0,Y 319.934,Z 172.634,A -85,B 0,C 180,E1 -15382.428,E2 -15382.428} C_VEL
LIN {X 0,Y 319.748,Z 172.653,A -85,B 0,C 180,E1 -15384.958,E2 -15384.958} C_VEL
LIN {X 0,Y 319.991,Z 172.623,A -85,B 0,C 180,E1 -15387.484,E2 -15387.484} C_VEL
LIN {X 0,Y 320.002,Z 172.622,A -85,B 0,C 180,E1 -15391.26,E2 -15391.26} C_VEL
LIN {X 0,Y 319.737,Z 172.659,A -85,B 0,C 180,E1 -15393.783,E2 -15393.783} C_VEL
LIN {X 0,Y 319.954,Z 172.628,A -85,B 0,C 180,E1 -15396.307,E2 -15396.307} C_VEL
LIN {X 0,Y 319.846,Z 172.641,A -85,B 0,C 180,E1 -15398.85,E2 -15398.85} C_VEL
LIN {X 0,Y 319.685,Z 172.661,A -85,B 0,C 180,E1 -15402.702,E2 -15402.702} C_VEL
LIN {X 0,Y 319.703,Z 172.662,A -85,B 0,C 180,E1 -15405.297,E2 -15405.297} C_VEL
LIN {X 0,Y 319.677,Z 172.666,A -85,B 0,C 180,E1 -15409.257,E2 -15409.257} C_VEL
LIN {X 0,Y 319.535,Z 172.684,A -85,B 0,C 180,E1 -15413.324,E2 -15413.324} C_VEL
LIN {X 0,Y 319.554,Z 172.677,A -85,B 0,C 180,E1 -15416.097,E2 -15416.097} C_VEL
LIN {X 0,Y 319.546,Z 172.683,A -85,B 0,C 180,E1 -15418.94,E2 -15418.94} C_VEL
LIN {X 0,Y 319.529,Z 172.68,A -85,B 0,C 180,E1 -15421.864,E2 -15421.864} C_VEL
LIN {X 0,Y 319.584,Z 172.674,A -85,B 0,C 180,E1 -15425.544,E2 -15425.544} C_VEL
LIN {X 0,Y 319.533,Z 172.68,A -85,B 0,C 180,E1 -15429.663,E2 -15429.663} C_VEL
LIN {X 0,Y 319.526,Z 172.681,A -85,B 0,C 180,E1 -15433.461,E2 -15433.461} C_VEL
LIN {X 0,Y 319.56,Z 172.677,A -85,B 0,C 180,E1 -15437.017,E2 -15437.017} C_VEL
LIN {X 0,Y 319.551,Z 172.683,A -85,B 0,C 180,E1 -15440.371,E2 -15440.371} C_VEL
LIN {X 0,Y 319.628,Z 172.671,A -85,B 0,C 180,E1 -15444.447,E2 -15444.447} C_VEL
LIN {X 0,Y 319.724,Z 172.878,A -85,B 0,C 180,E1 -15445.521,E2 -15445.521} C_VEL
LIN {X 0,Y 320.684,Z 178.656,A -85,B 0,C 180,E1 -15448.73,E2 -15448.73} C_VEL
LIN {X 0,Y 320.611,Z 181.866,A -85,B 0,C 180,E1 -15450.448,E2 -15450.448} C_VEL
LIN {X 0,Y 319.98,Z 189.115,A -85,B 0,C 180,E1 -15454.229,E2 -15454.229} C_VEL
LIN {X 0,Y 319.393,Z 196.533,A -85,B 0,C 180,E1 -15458.033,E2 -15458.033} C_VEL
LIN {X 0,Y 318.892,Z 204.429,A -85,B 0,C 180,E1 -15462.029,E2 -15462.029} C_VEL
LIN {X 0,Y 318.488,Z 212.707,A -85,B 0,C 180,E1 -15466.158,E2 -15466.158} C_VEL
LIN {X 0,Y 318.394,Z 215.27,A -85,B 0,C 180,E1 -15467.426,E2 -15467.426} C_VEL
LIN {X 0,Y 318.332,Z 216.918,A -85,B 0,C 180,E1 -15467.835,E2 -15467.835} C_VEL
LIN {X 0,Y 318.146,Z 220.237,A -85,B 0,C 180,E1 -15468.173,E2 -15468.173} C_VEL
LIN {X 0,Y 317.245,Z 226.816,A -85,B 0,C 180,E1 -15468.634,E2 -15468.634} C_VEL
LIN {X 0,Y 313.345,Z 238.647,A -85,B 0,C 180,E1 -15469.675,E2 -15469.675} C_VEL
LIN {X 0,Y 312.525,Z 242.546,A -85,B 0,C 180,E1 -15470.146,E2 -15470.146} C_VEL
LIN {X 0,Y 312.095,Z 251.98,A -85,B 0,C 180,E1 -15471.42,E2 -15471.42} C_VEL
LIN {X 0,Y 311.617,Z 260.714,A -85,B 0,C 180,E1 -15472.918,E2 -15472.918} C_VEL
LIN {X 0,Y 311.399,Z 267.973,A -85,B 0,C 180,E1 -15474.496,E2 -15474.496} C_VEL
LIN {X 0,Y 311.125,Z 273.808,A -85,B 0,C 180,E1 -15476.114,E2 -15476.114} C_VEL
LIN {X 0,Y 310.878,Z 279.033,A -85,B 0,C 180,E1 -15478.057,E2 -15478.057} C_VEL
LIN {X 0,Y 310.9,Z 282.624,A -85,B 0,C 180,E1 -15480,E2 -15480} C_VEL
LIN {X 0,Y 311.057,Z 284.178,A -85,B 0,C 180,E1 -15481.295,E2 -15481.295} C_VEL
LIN {X 0,Y 311.332,Z 285.1,A -85,B 0,C 180,E1 -15482.588,E2 -15482.588} C_VEL
LIN {X 0,Y 311.751,Z 285.378,A -85,B 0,C 180,E1 -15483.878,E2 -15483.878} C_VEL
LIN {X 0,Y 312.321,Z 285.022,A -85,B 0,C 180,E1 -15485.164,E2 -15485.164} C_VEL
LIN {X 0,Y 312.648,Z 284.097,A -85,B 0,C 180,E1 -15486.454,E2 -15486.454} C_VEL
LIN {X 0,Y 313.79,Z 281.519,A -85,B 0,C 180,E1 -15488.371,E2 -15488.371} C_VEL
LIN {X 0,Y 314.643,Z 279.005,A -85,B 0,C 180,E1 -15489.644,E2 -15489.644} C_VEL
LIN {X 0,Y 316.338,Z 273.899,A -85,B 0,C 180,E1 -15491.534,E2 -15491.534} C_VEL
LIN {X 0,Y 318.288,Z 267.632,A -85,B 0,C 180,E1 -15493.243,E2 -15493.243} C_VEL
LIN {X 0,Y 320.498,Z 259.586,A -85,B 0,C 180,E1 -15494.931,E2 -15494.931} C_VEL
LIN {X 0,Y 321.731,Z 254.729,A -85,B 0,C 180,E1 -15495.769,E2 -15495.769} C_VEL
LIN {X 0,Y 321.71,Z 246.942,A -85,B 0,C 180,E1 -15497.153,E2 -15497.153} C_VEL
LIN {X 0,Y 320.509,Z 237.373,A -85,B 0,C 180,E1 -15498.765,E2 -15498.765} C_VEL
LIN {X 0,Y 317.909,Z 226.648,A -85,B 0,C 180,E1 -15500.531,E2 -15500.531} C_VEL
LIN {X 0,Y 315.245,Z 218.397,A -85,B 0,C 180,E1 -15501.894,E2 -15501.894} C_VEL
LIN {X 0,Y 316.255,Z 214.061,A -85,B 0,C 180,E1 -15504.976,E2 -15504.976} C_VEL
LIN {X 0,Y 317.888,Z 208.79,A -85,B 0,C 180,E1 -15509.103,E2 -15509.103} C_VEL
LIN {X 0,Y 318.869,Z 205.756,A -85,B 0,C 180,E1 -15511.936,E2 -15511.936} C_VEL
LIN {X 0,Y 319.097,Z 204.451,A -85,B 0,C 180,E1 -15513.409,E2 -15513.409} C_VEL
LIN {X 0,Y 319.175,Z 202.999,A -85,B 0,C 180,E1 -15515.439,E2 -15515.439} C_VEL
LIN {X 0,Y 319.146,Z 201.629,A -85,B 0,C 180,E1 -15518.068,E2 -15518.068} C_VEL
LIN {X 0,Y 319.169,Z 200.638,A -85,B 0,C 180,E1 -15521.523,E2 -15521.523} C_VEL
LIN {X 0,Y 319.34,Z 200.695,A -85,B 0,C 180,E1 -15525.229,E2 -15525.229} C_VEL
LIN {X 0,Y 319.669,Z 201.854,A -85,B 0,C 180,E1 -15528.732,E2 -15528.732} C_VEL
LIN {X 0,Y 320.097,Z 204.164,A -85,B 0,C 180,E1 -15532.224,E2 -15532.224} C_VEL
LIN {X 0,Y 320.629,Z 207.047,A -85,B 0,C 180,E1 -15535.255,E2 -15535.255} C_VEL
LIN {X 0,Y 320.987,Z 208.825,A -85,B 0,C 180,E1 -15536.811,E2 -15536.811} C_VEL
LIN {X 0,Y 321.288,Z 211.12,A -85,B 0,C 180,E1 -15538.551,E2 -15538.551} C_VEL
LIN {X 0,Y 321.288,Z 213.024,A -85,B 0,C 180,E1 -15539.792,E2 -15539.792} C_VEL
LIN {X 0,Y 319.459,Z 218.171,A -85,B 0,C 180,E1 -15542.482,E2 -15542.482} C_VEL
LIN {X 0,Y 318.688,Z 220.574,A -85,B 0,C 180,E1 -15543.563,E2 -15543.563} C_VEL
LIN {X 0,Y 321.808,Z 232.237,A -85,B 0,C 180,E1 -15544.914,E2 -15544.914} C_VEL
LIN {X 0,Y 323.659,Z 242.79,A -85,B 0,C 180,E1 -15546.141,E2 -15546.141} C_VEL
LIN {X 0,Y 324.206,Z 251.834,A -85,B 0,C 180,E1 -15547.2,E2 -15547.2} C_VEL
LIN {X 0,Y 323.843,Z 257.407,A -85,B 0,C 180,E1 -15547.846,E2 -15547.846} C_VEL
LIN {X 0,Y 321.572,Z 268.593,A -85,B 0,C 180,E1 -15549.196,E2 -15549.196} C_VEL
LIN {X 0,Y 319.228,Z 278.634,A -85,B 0,C 180,E1 -15550.715,E2 -15550.715} C_VEL
LIN {X 0,Y 316.907,Z 287.965,A -85,B 0,C 180,E1 -15552.48,E2 -15552.48} C_VEL
LIN {X 0,Y 315.273,Z 295.018,A -85,B 0,C 180,E1 -15554.151,E2 -15554.151} C_VEL
LIN {X 0,Y 313.471,Z 302.575,A -85,B 0,C 180,E1 -15556.382,E2 -15556.382} C_VEL
LIN {X 0,Y 312.264,Z 307.652,A -85,B 0,C 180,E1 -15558.311,E2 -15558.311} C_VEL
LIN {X 0,Y 311.478,Z 311.608,A -85,B 0,C 180,E1 -15560.255,E2 -15560.255} C_VEL
LIN {X 0,Y 311.009,Z 314.54,A -85,B 0,C 180,E1 -15562.206,E2 -15562.206} C_VEL
LIN {X 0,Y 310.767,Z 316.973,A -85,B 0,C 180,E1 -15564.808,E2 -15564.808} C_VEL
LIN {X 0,Y 310.816,Z 317.545,A -85,B 0,C 180,E1 -15566.108,E2 -15566.108} C_VEL
LIN {X 0,Y 310.797,Z 317.695,A -85,B 0,C 180,E1 -15567.406,E2 -15567.406} C_VEL
LIN {X 0,Y 311.064,Z 317.462,A -85,B 0,C 180,E1 -15568.703,E2 -15568.703} C_VEL
LIN {X 0,Y 311.102,Z 316.746,A -85,B 0,C 180,E1 -15569.998,E2 -15569.998} C_VEL
LIN {X 0,Y 311.131,Z 315.59,A -85,B 0,C 180,E1 -15571.292,E2 -15571.292} C_VEL
LIN {X 0,Y 311.011,Z 312.966,A -85,B 0,C 180,E1 -15573.236,E2 -15573.236} C_VEL
LIN {X 0,Y 311.108,Z 309.234,A -85,B 0,C 180,E1 -15575.182,E2 -15575.182} C_VEL
LIN {X 0,Y 311.164,Z 304.205,A -85,B 0,C 180,E1 -15577.134,E2 -15577.134} C_VEL
LIN {X 0,Y 311.329,Z 297.698,A -85,B 0,C 180,E1 -15579.09,E2 -15579.09} C_VEL
LIN {X 0,Y 311.715,Z 289.482,A -85,B 0,C 180,E1 -15581.046,E2 -15581.046} C_VEL
LIN {X 0,Y 312.232,Z 280.902,A -85,B 0,C 180,E1 -15582.675,E2 -15582.675} C_VEL
LIN {X 0,Y 312.88,Z 271.464,A -85,B 0,C 180,E1 -15584.137,E2 -15584.137} C_VEL
LIN {X 0,Y 313.563,Z 261.336,A -85,B 0,C 180,E1 -15585.4,E2 -15585.4} C_VEL
LIN {X 0,Y 314.338,Z 249.522,A -85,B 0,C 180,E1 -15586.56,E2 -15586.56} C_VEL
LIN {X 0,Y 314.268,Z 244.338,A -85,B 0,C 180,E1 -15586.982,E2 -15586.982} C_VEL
LIN {X 0,Y 313.113,Z 231.895,A -85,B 0,C 180,E1 -15587.805,E2 -15587.805} C_VEL
LIN {X 0,Y 312.455,Z 220.14,A -85,B 0,C 180,E1 -15588.352,E2 -15588.352} C_VEL
LIN {X 0,Y 313.838,Z 207.945,A -85,B 0,C 180,E1 -15592.911,E2 -15592.911} C_VEL
LIN {X 0,Y 315.432,Z 197.195,A -85,B 0,C 180,E1 -15596.972,E2 -15596.972} C_VEL
LIN {X 0,Y 316.038,Z 193.027,A -85,B 0,C 180,E1 -15598.56,E2 -15598.56} C_VEL
LIN {X 0,Y 315.489,Z 188.836,A -85,B 0,C 180,E1 -15600.237,E2 -15600.237} C_VEL
LIN {X 0,Y 313.647,Z 179.672,A -85,B 0,C 180,E1 -15604.066,E2 -15604.066} C_VEL
LIN {X 0,Y 312.56,Z 173.556,A -85,B 0,C 180,E1 -15606.737,E2 -15606.737} C_VEL
LIN {X 0,Y 312.482,Z 173.563,A -85,B 0,C 180,E1 -15610.707,E2 -15610.707} C_VEL
LIN {X 0,Y 312.51,Z 173.557,A -85,B 0,C 180,E1 -15614.196,E2 -15614.196} C_VEL
LIN {X 0,Y 312.539,Z 173.552,A -85,B 0,C 180,E1 -15617.904,E2 -15617.904} C_VEL
LIN {X 0,Y 312.547,Z 173.552,A -85,B 0,C 180,E1 -15621.903,E2 -15621.903} C_VEL
LIN {X 0,Y 312.495,Z 173.558,A -85,B 0,C 180,E1 -15625.788,E2 -15625.788} C_VEL
LIN {X 0,Y 312.512,Z 173.554,A -85,B 0,C 180,E1 -15628.852,E2 -15628.852} C_VEL
LIN {X 0,Y 312.564,Z 173.552,A -85,B 0,C 180,E1 -15631.824,E2 -15631.824} C_VEL
LIN {X 0,Y 312.572,Z 173.547,A -85,B 0,C 180,E1 -15634.71,E2 -15634.71} C_VEL
LIN {X 0,Y 312.525,Z 173.553,A -85,B 0,C 180,E1 -15638.912,E2 -15638.912} C_VEL
LIN {X 0,Y 312.625,Z 173.545,A -85,B 0,C 180,E1 -15641.655,E2 -15641.655} C_VEL
LIN {X 0,Y 312.68,Z 173.537,A -85,B 0,C 180,E1 -15645.685,E2 -15645.685} C_VEL
LIN {X 0,Y 312.688,Z 173.535,A -85,B 0,C 180,E1 -15649.641,E2 -15649.641} C_VEL
LIN {X 0,Y 312.853,Z 173.512,A -85,B 0,C 180,E1 -15652.254,E2 -15652.254} C_VEL
LIN {X 0,Y 312.706,Z 173.533,A -85,B 0,C 180,E1 -15654.842,E2 -15654.842} C_VEL
LIN {X 0,Y 312.94,Z 173.503,A -85,B 0,C 180,E1 -15657.426,E2 -15657.426} C_VEL
LIN {X 0,Y 313.087,Z 173.482,A -85,B 0,C 180,E1 -15660,E2 -15660} C_VEL
LIN {X 0,Y 312.919,Z 173.506,A -85,B 0,C 180,E1 -15662.574,E2 -15662.574} C_VEL
LIN {X 0,Y 312.877,Z 173.509,A -85,B 0,C 180,E1 -15666.667,E2 -15666.667} C_VEL
LIN {X 0,Y 312.774,Z 173.524,A -85,B 0,C 180,E1 -15669.05,E2 -15669.05} C_VEL
LIN {X 0,Y 312.623,Z 173.542,A -85,B 0,C 180,E1 -15672.991,E2 -15672.991} C_VEL
LIN {X 0,Y 312.625,Z 173.54,A -85,B 0,C 180,E1 -15675.65,E2 -15675.65} C_VEL
LIN {X 0,Y 312.594,Z 173.545,A -85,B 0,C 180,E1 -15679.709,E2 -15679.709} C_VEL
LIN {X 0,Y 312.532,Z 173.553,A -85,B 0,C 180,E1 -15682.79,E2 -15682.79} C_VEL
LIN {X 0,Y 312.522,Z 173.556,A -85,B 0,C 180,E1 -15685.911,E2 -15685.911} C_VEL
LIN {X 0,Y 312.487,Z 173.56,A -85,B 0,C 180,E1 -15689.656,E2 -15689.656} C_VEL
LIN {X 0,Y 312.508,Z 173.558,A -85,B 0,C 180,E1 -15693.69,E2 -15693.69} C_VEL
LIN {X 0,Y 312.527,Z 173.555,A -85,B 0,C 180,E1 -15697.385,E2 -15697.385} C_VEL
LIN {X 0,Y 312.48,Z 173.558,A -85,B 0,C 180,E1 -15700.711,E2 -15700.711} C_VEL
LIN {X 0,Y 312.463,Z 173.561,A -85,B 0,C 180,E1 -15704.208,E2 -15704.208} C_VEL
LIN {X 0,Y 312.477,Z 173.56,A -85,B 0,C 180,E1 -15707.92,E2 -15707.92} C_VEL
LIN {X 0,Y 312.497,Z 173.557,A -85,B 0,C 180,E1 -15711.919,E2 -15711.919} C_VEL
LIN {X 0,Y 312.524,Z 173.553,A -85,B 0,C 180,E1 -15714.222,E2 -15714.222} C_VEL
LIN {X 0,Y 312.498,Z 173.559,A -85,B 0,C 180,E1 -15717.336,E2 -15717.336} C_VEL
LIN {X 0,Y 312.547,Z 173.552,A -85,B 0,C 180,E1 -15721.278,E2 -15721.278} C_VEL
LIN {X 0,Y 312.581,Z 173.55,A -85,B 0,C 180,E1 -15724.713,E2 -15724.713} C_VEL
LIN {X 0,Y 312.584,Z 173.545,A -85,B 0,C 180,E1 -15727.531,E2 -15727.531} C_VEL
LIN {X 0,Y 312.636,Z 173.539,A -85,B 0,C 180,E1 -15731.659,E2 -15731.659} C_VEL
LIN {X 0,Y 312.692,Z 173.532,A -85,B 0,C 180,E1 -15735.688,E2 -15735.688} C_VEL
LIN {X 0,Y 312.701,Z 173.531,A -85,B 0,C 180,E1 -15739.644,E2 -15739.644} C_VEL
LIN {X 0,Y 312.872,Z 173.515,A -85,B 0,C 180,E1 -15742.256,E2 -15742.256} C_VEL
LIN {X 0,Y 312.718,Z 173.529,A -85,B 0,C 180,E1 -15744.845,E2 -15744.845} C_VEL
LIN {X 0,Y 312.938,Z 173.502,A -85,B 0,C 180,E1 -15747.428,E2 -15747.428} C_VEL
LIN {X 0,Y 312.972,Z 173.498,A -85,B 0,C 180,E1 -15751.289,E2 -15751.289} C_VEL
LIN {X 0,Y 312.688,Z 173.537,A -85,B 0,C 180,E1 -15753.868,E2 -15753.868} C_VEL
LIN {X 0,Y 312.913,Z 173.505,A -85,B 0,C 180,E1 -15756.45,E2 -15756.45} C_VEL
LIN {X 0,Y 312.791,Z 173.52,A -85,B 0,C 180,E1 -15759.051,E2 -15759.051} C_VEL
LIN {X 0,Y 312.638,Z 173.539,A -85,B 0,C 180,E1 -15762.993,E2 -15762.993} C_VEL
LIN {X 0,Y 312.642,Z 173.542,A -85,B 0,C 180,E1 -15765.651,E2 -15765.651} C_VEL
LIN {X 0,Y 312.633,Z 173.544,A -85,B 0,C 180,E1 -15769.237,E2 -15769.237} C_VEL
LIN {X 0,Y 312.518,Z 173.555,A -85,B 0,C 180,E1 -15772.777,E2 -15772.777} C_VEL
LIN {X 0,Y 312.487,Z 173.56,A -85,B 0,C 180,E1 -15776.733,E2 -15776.733} C_VEL
LIN {X 0,Y 312.5,Z 173.556,A -85,B 0,C 180,E1 -15779.657,E2 -15779.657} C_VEL
LIN {X 0,Y 312.525,Z 173.553,A -85,B 0,C 180,E1 -15783.69,E2 -15783.69} C_VEL
LIN {X 0,Y 312.518,Z 173.554,A -85,B 0,C 180,E1 -15787.388,E2 -15787.388} C_VEL
LIN {X 0,Y 312.446,Z 173.567,A -85,B 0,C 180,E1 -15790.718,E2 -15790.718} C_VEL
LIN {X 0,Y 312.457,Z 173.564,A -85,B 0,C 180,E1 -15794.211,E2 -15794.211} C_VEL
LIN {X 0,Y 312.518,Z 173.555,A -85,B 0,C 180,E1 -15797.914,E2 -15797.914} C_VEL
LIN {X 0,Y 312.492,Z 173.559,A -85,B 0,C 180,E1 -15801.923,E2 -15801.923} C_VEL
LIN {X 0,Y 312.653,Z 173.592,A -85,B 0,C 180,E1 -15805.32,E2 -15805.32} C_VEL
LIN {X 0,Y 313.576,Z 178.991,A -85,B 0,C 180,E1 -15808.397,E2 -15808.397} C_VEL
LIN {X 0,Y 313.547,Z 182.769,A -85,B 0,C 180,E1 -15810.454,E2 -15810.454} C_VEL
LIN {X 0,Y 312.948,Z 189.331,A -85,B 0,C 180,E1 -15813.938,E2 -15813.938} C_VEL
LIN {X 0,Y 312.292,Z 197.492,A -85,B 0,C 180,E1 -15818.203,E2 -15818.203} C_VEL
LIN {X 0,Y 311.783,Z 205.414,A -85,B 0,C 180,E1 -15822.284,E2 -15822.284} C_VEL
LIN {X 0,Y 311.411,Z 212.809,A -85,B 0,C 180,E1 -15826.038,E2 -15826.038} C_VEL
LIN {X 0,Y 311.287,Z 216.346,A -85,B 0,C 180,E1 -15827.822,E2 -15827.822} C_VEL
LIN {X 0,Y 312.161,Z 229.454,A -85,B 0,C 180,E1 -15828.803,E2 -15828.803} C_VEL
LIN {X 0,Y 312.819,Z 238.129,A -85,B 0,C 180,E1 -15829.646,E2 -15829.646} C_VEL
LIN {X 0,Y 312.525,Z 242.546,A -85,B 0,C 180,E1 -15830.146,E2 -15830.146} C_VEL
LIN {X 0,Y 311.578,Z 247.372,A -85,B 0,C 180,E1 -15830.755,E2 -15830.755} C_VEL
LIN {X 0,Y 308.302,Z 254.702,A -85,B 0,C 180,E1 -15831.836,E2 -15831.836} C_VEL
LIN {X 0,Y 305.125,Z 261.447,A -85,B 0,C 180,E1 -15833.064,E2 -15833.064} C_VEL
LIN {X 0,Y 304.345,Z 265.309,A -85,B 0,C 180,E1 -15833.895,E2 -15833.895} C_VEL
LIN {X 0,Y 304.133,Z 272.288,A -85,B 0,C 180,E1 -15835.693,E2 -15835.693} C_VEL
LIN {X 0,Y 303.843,Z 277.241,A -85,B 0,C 180,E1 -15837.349,E2 -15837.349} C_VEL
LIN {X 0,Y 303.764,Z 281.574,A -85,B 0,C 180,E1 -15839.337,E2 -15839.337} C_VEL
LIN {X 0,Y 303.962,Z 284.363,A -85,B 0,C 180,E1 -15841.325,E2 -15841.325} C_VEL
LIN {X 0,Y 304.247,Z 285.412,A -85,B 0,C 180,E1 -15842.648,E2 -15842.648} C_VEL
LIN {X 0,Y 304.699,Z 285.842,A -85,B 0,C 180,E1 -15843.968,E2 -15843.968} C_VEL
LIN {X 0,Y 305.289,Z 285.656,A -85,B 0,C 180,E1 -15845.284,E2 -15845.284} C_VEL
LIN {X 0,Y 305.659,Z 284.903,A -85,B 0,C 180,E1 -15846.602,E2 -15846.602} C_VEL
LIN {X 0,Y 306.863,Z 282.564,A -85,B 0,C 180,E1 -15848.561,E2 -15848.561} C_VEL
LIN {X 0,Y 308.33,Z 278.809,A -85,B 0,C 180,E1 -15850.507,E2 -15850.507} C_VEL
LIN {X 0,Y 310.251,Z 273.485,A -85,B 0,C 180,E1 -15852.427,E2 -15852.427} C_VEL
LIN {X 0,Y 312.176,Z 267.677,A -85,B 0,C 180,E1 -15854.006,E2 -15854.006} C_VEL
LIN {X 0,Y 314.345,Z 260.419,A -85,B 0,C 180,E1 -15855.563,E2 -15855.563} C_VEL
LIN {X 0,Y 315.488,Z 255.738,A -85,B 0,C 180,E1 -15856.416,E2 -15856.416} C_VEL
LIN {X 0,Y 315.535,Z 248.207,A -85,B 0,C 180,E1 -15857.834,E2 -15857.834} C_VEL
LIN {X 0,Y 314.346,Z 238.46,A -85,B 0,C 180,E1 -15859.595,E2 -15859.595} C_VEL
LIN {X 0,Y 312.017,Z 228.717,A -85,B 0,C 180,E1 -15861.334,E2 -15861.334} C_VEL
LIN {X 0,Y 309.51,Z 221.258,A -85,B 0,C 180,E1 -15862.707,E2 -15862.707} C_VEL
LIN {X 0,Y 308.782,Z 218.505,A -85,B 0,C 180,E1 -15863.206,E2 -15863.206} C_VEL
LIN {X 0,Y 310.166,Z 213.614,A -85,B 0,C 180,E1 -15866.948,E2 -15866.948} C_VEL
LIN {X 0,Y 311.341,Z 210.3,A -85,B 0,C 180,E1 -15869.776,E2 -15869.776} C_VEL
LIN {X 0,Y 311.889,Z 208.785,A -85,B 0,C 180,E1 -15871.217,E2 -15871.217} C_VEL
LIN {X 0,Y 312.428,Z 206.638,A -85,B 0,C 180,E1 -15873.661,E2 -15873.661} C_VEL
LIN {X 0,Y 312.484,Z 205.17,A -85,B 0,C 180,E1 -15875.934,E2 -15875.934} C_VEL
LIN {X 0,Y 312.488,Z 203.789,A -85,B 0,C 180,E1 -15879.031,E2 -15879.031} C_VEL
LIN {X 0,Y 312.551,Z 203.163,A -85,B 0,C 180,E1 -15882.422,E2 -15882.422} C_VEL
LIN {X 0,Y 312.803,Z 203.484,A -85,B 0,C 180,E1 -15885.97,E2 -15885.97} C_VEL
LIN {X 0,Y 313.127,Z 204.828,A -85,B 0,C 180,E1 -15889.389,E2 -15889.389} C_VEL
LIN {X 0,Y 313.527,Z 207.162,A -85,B 0,C 180,E1 -15892.753,E2 -15892.753} C_VEL
LIN {X 0,Y 314.107,Z 210.238,A -85,B 0,C 180,E1 -15895.88,E2 -15895.88} C_VEL
LIN {X 0,Y 314.529,Z 212.95,A -85,B 0,C 180,E1 -15898.114,E2 -15898.114} C_VEL
LIN {X 0,Y 314.483,Z 215.444,A -85,B 0,C 180,E1 -15899.811,E2 -15899.811} C_VEL
LIN {X 0,Y 312.603,Z 220.526,A -85,B 0,C 180,E1 -15902.441,E2 -15902.441} C_VEL
LIN {X 0,Y 313.657,Z 224.153,A -85,B 0,C 180,E1 -15902.9,E2 -15902.9} C_VEL
LIN {X 0,Y 316.702,Z 236.936,A -85,B 0,C 180,E1 -15904.521,E2 -15904.521} C_VEL
LIN {X 0,Y 318.035,Z 247.281,A -85,B 0,C 180,E1 -15905.818,E2 -15905.818} C_VEL
LIN {X 0,Y 318.1,Z 255.963,A -85,B 0,C 180,E1 -15906.909,E2 -15906.909} C_VEL
LIN {X 0,Y 316.395,Z 264.889,A -85,B 0,C 180,E1 -15907.984,E2 -15907.984} C_VEL
LIN {X 0,Y 313.579,Z 276.453,A -85,B 0,C 180,E1 -15909.67,E2 -15909.67} C_VEL
LIN {X 0,Y 310.887,Z 286.466,A -85,B 0,C 180,E1 -15911.547,E2 -15911.547} C_VEL
LIN {X 0,Y 309.027,Z 293.336,A -85,B 0,C 180,E1 -15913.142,E2 -15913.142} C_VEL
LIN {X 0,Y 307.406,Z 300.095,A -85,B 0,C 180,E1 -15915.094,E2 -15915.094} C_VEL
LIN {X 0,Y 305.631,Z 306.364,A -85,B 0,C 180,E1 -15917.38,E2 -15917.38} C_VEL
LIN {X 0,Y 304.692,Z 310.506,A -85,B 0,C 180,E1 -15919.364,E2 -15919.364} C_VEL
LIN {X 0,Y 304.252,Z 312.676,A -85,B 0,C 180,E1 -15920.693,E2 -15920.693} C_VEL
LIN {X 0,Y 303.748,Z 315.748,A -85,B 0,C 180,E1 -15923.355,E2 -15923.355} C_VEL
LIN {X 0,Y 303.688,Z 316.642,A -85,B 0,C 180,E1 -15924.687,E2 -15924.687} C_VEL
LIN {X 0,Y 303.745,Z 317.128,A -85,B 0,C 180,E1 -15926.018,E2 -15926.018} C_VEL
LIN {X 0,Y 303.716,Z 317.209,A -85,B 0,C 180,E1 -15927.345,E2 -15927.345} C_VEL
LIN {X 0,Y 304,Z 316.861,A -85,B 0,C 180,E1 -15928.673,E2 -15928.673} C_VEL
LIN {X 0,Y 304.047,Z 316.059,A -85,B 0,C 180,E1 -15929.998,E2 -15929.998} C_VEL
LIN {X 0,Y 304.076,Z 314.837,A -85,B 0,C 180,E1 -15931.322,E2 -15931.322} C_VEL
LIN {X 0,Y 303.951,Z 312.06,A -85,B 0,C 180,E1 -15933.312,E2 -15933.312} C_VEL
LIN {X 0,Y 304.061,Z 308.132,A -85,B 0,C 180,E1 -15935.303,E2 -15935.303} C_VEL
LIN {X 0,Y 304.129,Z 302.9,A -85,B 0,C 180,E1 -15937.3,E2 -15937.3} C_VEL
LIN {X 0,Y 304.305,Z 296.206,A -85,B 0,C 180,E1 -15939.301,E2 -15939.301} C_VEL
LIN {X 0,Y 304.745,Z 287.665,A -85,B 0,C 180,E1 -15941.302,E2 -15941.302} C_VEL
LIN {X 0,Y 305.263,Z 278.817,A -85,B 0,C 180,E1 -15942.97,E2 -15942.97} C_VEL
LIN {X 0,Y 305.841,Z 270.155,A -85,B 0,C 180,E1 -15944.299,E2 -15944.299} C_VEL
LIN {X 0,Y 306.719,Z 258.182,A -85,B 0,C 180,E1 -15945.768,E2 -15945.768} C_VEL
LIN {X 0,Y 307.348,Z 246.567,A -85,B 0,C 180,E1 -15946.863,E2 -15946.863} C_VEL
LIN {X 0,Y 306.146,Z 233.723,A -85,B 0,C 180,E1 -15947.792,E2 -15947.792} C_VEL
LIN {X 0,Y 305.417,Z 221.618,A -85,B 0,C 180,E1 -15948.4,E2 -15948.4} C_VEL
LIN {X 0,Y 305.407,Z 220.061,A -85,B 0,C 180,E1 -15948.487,E2 -15948.487} C_VEL
LIN {X 0,Y 306.908,Z 207.5,A -85,B 0,C 180,E1 -15953.318,E2 -15953.318} C_VEL
LIN {X 0,Y 308.753,Z 195.834,A -85,B 0,C 180,E1 -15957.849,E2 -15957.849} C_VEL
LIN {X 0,Y 308.894,Z 192.246,A -85,B 0,C 180,E1 -15959.28,E2 -15959.28} C_VEL
LIN {X 0,Y 307.027,Z 182.652,A -85,B 0,C 180,E1 -15963.321,E2 -15963.321} C_VEL
LIN {X 0,Y 305.507,Z 174.434,A -85,B 0,C 180,E1 -15966.938,E2 -15966.938} C_VEL
LIN {X 0,Y 305.447,Z 174.439,A -85,B 0,C 180,E1 -15970.598,E2 -15970.598} C_VEL
LIN {X 0,Y 305.452,Z 174.439,A -85,B 0,C 180,E1 -15974.499,E2 -15974.499} C_VEL
LIN {X 0,Y 305.485,Z 174.432,A -85,B 0,C 180,E1 -15978.15,E2 -15978.15} C_VEL
LIN {X 0,Y 305.509,Z 174.427,A -85,B 0,C 180,E1 -15981.602,E2 -15981.602} C_VEL
LIN {X 0,Y 305.452,Z 174.434,A -85,B 0,C 180,E1 -15984.885,E2 -15984.885} C_VEL
LIN {X 0,Y 305.441,Z 174.438,A -85,B 0,C 180,E1 -15988.353,E2 -15988.353} C_VEL
LIN {X 0,Y 305.509,Z 174.427,A -85,B 0,C 180,E1 -15991.112,E2 -15991.112} C_VEL
LIN {X 0,Y 305.559,Z 174.423,A -85,B 0,C 180,E1 -15994.087,E2 -15994.087} C_VEL
LIN {X 0,Y 305.469,Z 174.432,A -85,B 0,C 180,E1 -15998.4,E2 -15998.4} C_VEL
LIN {X 0,Y 305.576,Z 174.42,A -85,B 0,C 180,E1 -16001.217,E2 -16001.217} C_VEL
LIN {X 0,Y 305.636,Z 174.415,A -85,B 0,C 180,E1 -16005.348,E2 -16005.348} C_VEL
LIN {X 0,Y 305.626,Z 174.417,A -85,B 0,C 180,E1 -16009.399,E2 -16009.399} C_VEL
LIN {X 0,Y 305.795,Z 174.391,A -85,B 0,C 180,E1 -16012.074,E2 -16012.074} C_VEL
LIN {X 0,Y 305.677,Z 174.407,A -85,B 0,C 180,E1 -16014.723,E2 -16014.723} C_VEL
LIN {X 0,Y 305.947,Z 174.374,A -85,B 0,C 180,E1 -16018.684,E2 -16018.684} C_VEL
LIN {X 0,Y 305.942,Z 174.375,A -85,B 0,C 180,E1 -16021.316,E2 -16021.316} C_VEL
LIN {X 0,Y 305.833,Z 174.389,A -85,B 0,C 180,E1 -16026.646,E2 -16026.646} C_VEL
LIN {X 0,Y 305.722,Z 174.401,A -85,B 0,C 180,E1 -16029.26,E2 -16029.26} C_VEL
LIN {X 0,Y 305.577,Z 174.419,A -85,B 0,C 180,E1 -16033.296,E2 -16033.296} C_VEL
LIN {X 0,Y 305.58,Z 174.419,A -85,B 0,C 180,E1 -16036.021,E2 -16036.021} C_VEL
LIN {X 0,Y 305.568,Z 174.419,A -85,B 0,C 180,E1 -16039.448,E2 -16039.448} C_VEL
LIN {X 0,Y 305.475,Z 174.431,A -85,B 0,C 180,E1 -16043.041,E2 -16043.041} C_VEL
LIN {X 0,Y 305.462,Z 174.437,A -85,B 0,C 180,E1 -16046.2,E2 -16046.2} C_VEL
LIN {X 0,Y 305.445,Z 174.435,A -85,B 0,C 180,E1 -16049.038,E2 -16049.038} C_VEL
LIN {X 0,Y 305.424,Z 174.442,A -85,B 0,C 180,E1 -16051.954,E2 -16051.954} C_VEL
LIN {X 0,Y 305.451,Z 174.434,A -85,B 0,C 180,E1 -16055.115,E2 -16055.115} C_VEL
LIN {X 0,Y 305.457,Z 174.433,A -85,B 0,C 180,E1 -16058.535,E2 -16058.535} C_VEL
LIN {X 0,Y 305.467,Z 174.431,A -85,B 0,C 180,E1 -16062.592,E2 -16062.592} C_VEL
LIN {X 0,Y 305.434,Z 174.436,A -85,B 0,C 180,E1 -16066.35,E2 -16066.35} C_VEL
LIN {X 0,Y 305.45,Z 174.435,A -85,B 0,C 180,E1 -16069.894,E2 -16069.894} C_VEL
LIN {X 0,Y 305.473,Z 174.433,A -85,B 0,C 180,E1 -16073.634,E2 -16073.634} C_VEL
LIN {X 0,Y 305.458,Z 174.434,A -85,B 0,C 180,E1 -16076.485,E2 -16076.485} C_VEL
LIN {X 0,Y 305.491,Z 174.433,A -85,B 0,C 180,E1 -16080.952,E2 -16080.952} C_VEL
LIN {X 0,Y 305.567,Z 174.42,A -85,B 0,C 180,E1 -16084.09,E2 -16084.09} C_VEL
LIN {X 0,Y 305.498,Z 174.43,A -85,B 0,C 180,E1 -16088.405,E2 -16088.405} C_VEL
LIN {X 0,Y 305.587,Z 174.418,A -85,B 0,C 180,E1 -16091.22,E2 -16091.22} C_VEL
LIN {X 0,Y 305.647,Z 174.409,A -85,B 0,C 180,E1 -16095.351,E2 -16095.351} C_VEL
LIN {X 0,Y 305.638,Z 174.41,A -85,B 0,C 180,E1 -16099.402,E2 -16099.402} C_VEL
LIN {X 0,Y 305.813,Z 174.392,A -85,B 0,C 180,E1 -16102.077,E2 -16102.077} C_VEL
LIN {X 0,Y 305.69,Z 174.405,A -85,B 0,C 180,E1 -16104.726,E2 -16104.726} C_VEL
LIN {X 0,Y 305.942,Z 174.373,A -85,B 0,C 180,E1 -16108.686,E2 -16108.686} C_VEL
LIN {X 0,Y 305.883,Z 174.38,A -85,B 0,C 180,E1 -16112.636,E2 -16112.636} C_VEL
LIN {X 0,Y 305.855,Z 174.384,A -85,B 0,C 180,E1 -16116.599,E2 -16116.599} C_VEL
LIN {X 0,Y 305.739,Z 174.4,A -85,B 0,C 180,E1 -16119.262,E2 -16119.262} C_VEL
LIN {X 0,Y 305.592,Z 174.419,A -85,B 0,C 180,E1 -16123.298,E2 -16123.298} C_VEL
LIN {X 0,Y 305.598,Z 174.417,A -85,B 0,C 180,E1 -16126.022,E2 -16126.022} C_VEL
LIN {X 0,Y 305.579,Z 174.422,A -85,B 0,C 180,E1 -16129.446,E2 -16129.446} C_VEL
LIN {X 0,Y 305.459,Z 174.436,A -85,B 0,C 180,E1 -16133.027,E2 -16133.027} C_VEL
LIN {X 0,Y 305.455,Z 174.433,A -85,B 0,C 180,E1 -16136.192,E2 -16136.192} C_VEL
LIN {X 0,Y 305.452,Z 174.438,A -85,B 0,C 180,E1 -16139.035,E2 -16139.035} C_VEL
LIN {X 0,Y 305.441,Z 174.435,A -85,B 0,C 180,E1 -16141.954,E2 -16141.954} C_VEL
LIN {X 0,Y 305.467,Z 174.435,A -85,B 0,C 180,E1 -16145.115,E2 -16145.115} C_VEL
LIN {X 0,Y 305.438,Z 174.439,A -85,B 0,C 180,E1 -16148.526,E2 -16148.526} C_VEL
LIN {X 0,Y 305.441,Z 174.44,A -85,B 0,C 180,E1 -16152.583,E2 -16152.583} C_VEL
LIN {X 0,Y 305.435,Z 174.44,A -85,B 0,C 180,E1 -16156.347,E2 -16156.347} C_VEL
LIN {X 0,Y 305.463,Z 174.434,A -85,B 0,C 180,E1 -16159.893,E2 -16159.893} C_VEL
LIN {X 0,Y 305.518,Z 174.426,A -85,B 0,C 180,E1 -16163.625,E2 -16163.625} C_VEL
LIN {X 0,Y 305.637,Z 174.585,A -85,B 0,C 180,E1 -16165.295,E2 -16165.295} C_VEL
LIN {X 0,Y 306.482,Z 179.575,A -85,B 0,C 180,E1 -16168.169,E2 -16168.169} C_VEL
LIN {X 0,Y 306.63,Z 182.33,A -85,B 0,C 180,E1 -16169.719,E2 -16169.719} C_VEL
LIN {X 0,Y 305.928,Z 189.534,A -85,B 0,C 180,E1 -16173.632,E2 -16173.632} C_VEL
LIN {X 0,Y 305.299,Z 197.143,A -85,B 0,C 180,E1 -16177.699,E2 -16177.699} C_VEL
LIN {X 0,Y 304.761,Z 205.055,A -85,B 0,C 180,E1 -16181.861,E2 -16181.861} C_VEL
LIN {X 0,Y 304.336,Z 212.862,A -85,B 0,C 180,E1 -16185.913,E2 -16185.913} C_VEL
LIN {X 0,Y 304.228,Z 216.421,A -85,B 0,C 180,E1 -16187.746,E2 -16187.746} C_VEL
LIN {X 0,Y 304.961,Z 228.111,A -85,B 0,C 180,E1 -16188.619,E2 -16188.619} C_VEL
LIN {X 0,Y 305.744,Z 237.87,A -85,B 0,C 180,E1 -16189.571,E2 -16189.571} C_VEL
LIN {X 0,Y 305.174,Z 248.5,A -85,B 0,C 180,E1 -16190.89,E2 -16190.89} C_VEL
LIN {X 0,Y 304.701,Z 257.817,A -85,B 0,C 180,E1 -16192.379,E2 -16192.379} C_VEL
LIN {X 0,Y 304.345,Z 265.309,A -85,B 0,C 180,E1 -16193.895,E2 -16193.895} C_VEL
LIN {X 0,Y 303.571,Z 268.916,A -85,B 0,C 180,E1 -16194.766,E2 -16194.766} C_VEL
LIN {X 0,Y 301.849,Z 272.15,A -85,B 0,C 180,E1 -16195.654,E2 -16195.654} C_VEL
LIN {X 0,Y 297.879,Z 277.63,A -85,B 0,C 180,E1 -16197.543,E2 -16197.543} C_VEL
LIN {X 0,Y 296.764,Z 279.984,A -85,B 0,C 180,E1 -16198.576,E2 -16198.576} C_VEL
LIN {X 0,Y 296.672,Z 280.696,A -85,B 0,C 180,E1 -16198.933,E2 -16198.933} C_VEL
LIN {X 0,Y 296.711,Z 282.633,A -85,B 0,C 180,E1 -16200,E2 -16200} C_VEL
LIN {X 0,Y 296.869,Z 284.484,A -85,B 0,C 180,E1 -16201.357,E2 -16201.357} C_VEL
LIN {X 0,Y 297.161,Z 285.703,A -85,B 0,C 180,E1 -16202.711,E2 -16202.711} C_VEL
LIN {X 0,Y 297.632,Z 286.3,A -85,B 0,C 180,E1 -16204.062,E2 -16204.062} C_VEL
LIN {X 0,Y 298.261,Z 286.26,A -85,B 0,C 180,E1 -16205.408,E2 -16205.408} C_VEL
LIN {X 0,Y 298.673,Z 285.651,A -85,B 0,C 180,E1 -16206.757,E2 -16206.757} C_VEL
LIN {X 0,Y 299.405,Z 284.439,A -85,B 0,C 180,E1 -16208.097,E2 -16208.097} C_VEL
LIN {X 0,Y 300.889,Z 281.472,A -85,B 0,C 180,E1 -16210.089,E2 -16210.089} C_VEL
LIN {X 0,Y 302.727,Z 277.026,A -85,B 0,C 180,E1 -16212.06,E2 -16212.06} C_VEL
LIN {X 0,Y 305.072,Z 270.92,A -85,B 0,C 180,E1 -16213.998,E2 -16213.998} C_VEL
LIN {X 0,Y 307.294,Z 264.384,A -85,B 0,C 180,E1 -16215.589,E2 -16215.589} C_VEL
LIN {X 0,Y 309.225,Z 257.639,A -85,B 0,C 180,E1 -16216.93,E2 -16216.93} C_VEL
LIN {X 0,Y 309.394,Z 249.656,A -85,B 0,C 180,E1 -16218.543,E2 -16218.543} C_VEL
LIN {X 0,Y 308.432,Z 240.512,A -85,B 0,C 180,E1 -16220.311,E2 -16220.311} C_VEL
LIN {X 0,Y 306.492,Z 231.52,A -85,B 0,C 180,E1 -16222.036,E2 -16222.036} C_VEL
LIN {X 0,Y 303.985,Z 223.142,A -85,B 0,C 180,E1 -16223.685,E2 -16223.685} C_VEL
LIN {X 0,Y 302.768,Z 220.166,A -85,B 0,C 180,E1 -16224.332,E2 -16224.332} C_VEL
LIN {X 0,Y 302.463,Z 218.639,A -85,B 0,C 180,E1 -16224.633,E2 -16224.633} C_VEL
LIN {X 0,Y 304.22,Z 213.403,A -85,B 0,C 180,E1 -16229.022,E2 -16229.022} C_VEL
LIN {X 0,Y 305.322,Z 210.439,A -85,B 0,C 180,E1 -16231.967,E2 -16231.967} C_VEL
LIN {X 0,Y 305.754,Z 208.706,A -85,B 0,C 180,E1 -16234.156,E2 -16234.156} C_VEL
LIN {X 0,Y 305.823,Z 207.237,A -85,B 0,C 180,E1 -16236.691,E2 -16236.691} C_VEL
LIN {X 0,Y 305.867,Z 206.452,A -85,B 0,C 180,E1 -16238.624,E2 -16238.624} C_VEL
LIN {X 0,Y 305.909,Z 205.801,A -85,B 0,C 180,E1 -16241.779,E2 -16241.779} C_VEL
LIN {X 0,Y 306.125,Z 205.97,A -85,B 0,C 180,E1 -16245.373,E2 -16245.373} C_VEL
LIN {X 0,Y 306.379,Z 206.916,A -85,B 0,C 180,E1 -16248.298,E2 -16248.298} C_VEL
LIN {X 0,Y 306.801,Z 208.988,A -85,B 0,C 180,E1 -16251.791,E2 -16251.791} C_VEL
LIN {X 0,Y 307.371,Z 212.197,A -85,B 0,C 180,E1 -16255.4,E2 -16255.4} C_VEL
LIN {X 0,Y 307.855,Z 215.667,A -85,B 0,C 180,E1 -16258.325,E2 -16258.325} C_VEL
LIN {X 0,Y 307.639,Z 217.861,A -85,B 0,C 180,E1 -16259.827,E2 -16259.827} C_VEL
LIN {X 0,Y 306.603,Z 220.32,A -85,B 0,C 180,E1 -16261.184,E2 -16261.184} C_VEL
LIN {X 0,Y 310.028,Z 233.595,A -85,B 0,C 180,E1 -16263.037,E2 -16263.037} C_VEL
LIN {X 0,Y 311.906,Z 245.375,A -85,B 0,C 180,E1 -16264.65,E2 -16264.65} C_VEL
LIN {X 0,Y 312.228,Z 254.133,A -85,B 0,C 180,E1 -16265.828,E2 -16265.828} C_VEL
LIN {X 0,Y 311.744,Z 259.916,A -85,B 0,C 180,E1 -16266.586,E2 -16266.586} C_VEL
LIN {X 0,Y 308.906,Z 271.318,A -85,B 0,C 180,E1 -16268.125,E2 -16268.125} C_VEL
LIN {X 0,Y 306.576,Z 279.781,A -85,B 0,C 180,E1 -16269.536,E2 -16269.536} C_VEL
LIN {X 0,Y 303.823,Z 289.066,A -85,B 0,C 180,E1 -16271.469,E2 -16271.469} C_VEL
LIN {X 0,Y 301.738,Z 296.485,A -85,B 0,C 180,E1 -16273.42,E2 -16273.42} C_VEL
LIN {X 0,Y 299.71,Z 303.419,A -85,B 0,C 180,E1 -16275.744,E2 -16275.744} C_VEL
LIN {X 0,Y 298.316,Z 308.09,A -85,B 0,C 180,E1 -16277.757,E2 -16277.757} C_VEL
LIN {X 0,Y 297.431,Z 311.688,A -85,B 0,C 180,E1 -16279.79,E2 -16279.79} C_VEL
LIN {X 0,Y 296.885,Z 314.295,A -85,B 0,C 180,E1 -16281.832,E2 -16281.832} C_VEL
LIN {X 0,Y 296.627,Z 316.195,A -85,B 0,C 180,E1 -16284.334,E2 -16284.334} C_VEL
LIN {X 0,Y 296.651,Z 316.71,A -85,B 0,C 180,E1 -16285.922,E2 -16285.922} C_VEL
LIN {X 0,Y 296.638,Z 316.669,A -85,B 0,C 180,E1 -16287.282,E2 -16287.282} C_VEL
LIN {X 0,Y 296.936,Z 316.228,A -85,B 0,C 180,E1 -16288.642,E2 -16288.642} C_VEL
LIN {X 0,Y 296.994,Z 315.36,A -85,B 0,C 180,E1 -16289.998,E2 -16289.998} C_VEL
LIN {X 0,Y 297.022,Z 314.005,A -85,B 0,C 180,E1 -16291.354,E2 -16291.354} C_VEL
LIN {X 0,Y 296.914,Z 311.057,A -85,B 0,C 180,E1 -16293.39,E2 -16293.39} C_VEL
LIN {X 0,Y 297.018,Z 306.964,A -85,B 0,C 180,E1 -16295.429,E2 -16295.429} C_VEL
LIN {X 0,Y 297.095,Z 301.56,A -85,B 0,C 180,E1 -16297.473,E2 -16297.473} C_VEL
LIN {X 0,Y 297.301,Z 294.587,A -85,B 0,C 180,E1 -16299.523,E2 -16299.523} C_VEL
LIN {X 0,Y 297.771,Z 285.781,A -85,B 0,C 180,E1 -16301.571,E2 -16301.571} C_VEL
LIN {X 0,Y 298.45,Z 275.49,A -85,B 0,C 180,E1 -16303.444,E2 -16303.444} C_VEL
LIN {X 0,Y 299.102,Z 264.87,A -85,B 0,C 180,E1 -16304.977,E2 -16304.977} C_VEL
LIN {X 0,Y 299.861,Z 254.842,A -85,B 0,C 180,E1 -16306.133,E2 -16306.133} C_VEL
LIN {X 0,Y 300.227,Z 246.408,A -85,B 0,C 180,E1 -16306.924,E2 -16306.924} C_VEL
LIN {X 0,Y 299.042,Z 233.609,A -85,B 0,C 180,E1 -16307.875,E2 -16307.875} C_VEL
LIN {X 0,Y 298.339,Z 221.618,A -85,B 0,C 180,E1 -16308.496,E2 -16308.496} C_VEL
LIN {X 0,Y 298.321,Z 220.038,A -85,B 0,C 180,E1 -16308.586,E2 -16308.586} C_VEL
LIN {X 0,Y 299.867,Z 207.695,A -85,B 0,C 180,E1 -16313.477,E2 -16313.477} C_VEL
LIN {X 0,Y 301.627,Z 196.905,A -85,B 0,C 180,E1 -16317.773,E2 -16317.773} C_VEL
LIN {X 0,Y 301.879,Z 193.242,A -85,B 0,C 180,E1 -16319.265,E2 -16319.265} C_VEL
LIN {X 0,Y 300.342,Z 185.518,A -85,B 0,C 180,E1 -16322.605,E2 -16322.605} C_VEL
LIN {X 0,Y 298.577,Z 176.041,A -85,B 0,C 180,E1 -16326.841,E2 -16326.841} C_VEL
LIN {X 0,Y 298.459,Z 175.311,A -85,B 0,C 180,E1 -16327.231,E2 -16327.231} C_VEL
LIN {X 0,Y 298.377,Z 175.316,A -85,B 0,C 180,E1 -16331.259,E2 -16331.259} C_VEL
LIN {X 0,Y 298.408,Z 175.312,A -85,B 0,C 180,E1 -16335.045,E2 -16335.045} C_VEL
LIN {X 0,Y 298.442,Z 175.309,A -85,B 0,C 180,E1 -16338.748,E2 -16338.748} C_VEL
LIN {X 0,Y 298.46,Z 175.305,A -85,B 0,C 180,E1 -16343.185,E2 -16343.185} C_VEL
LIN {X 0,Y 298.384,Z 175.314,A -85,B 0,C 180,E1 -16347.198,E2 -16347.198} C_VEL
LIN {X 0,Y 298.42,Z 175.31,A -85,B 0,C 180,E1 -16350.613,E2 -16350.613} C_VEL
LIN {X 0,Y 298.473,Z 175.305,A -85,B 0,C 180,E1 -16353.472,E2 -16353.472} C_VEL
LIN {X 0,Y 298.418,Z 175.31,A -85,B 0,C 180,E1 -16356.698,E2 -16356.698} C_VEL
LIN {X 0,Y 298.525,Z 175.297,A -85,B 0,C 180,E1 -16360.756,E2 -16360.756} C_VEL
LIN {X 0,Y 298.58,Z 175.291,A -85,B 0,C 180,E1 -16364.994,E2 -16364.994} C_VEL
LIN {X 0,Y 298.581,Z 175.293,A -85,B 0,C 180,E1 -16369.146,E2 -16369.146} C_VEL
LIN {X 0,Y 298.741,Z 175.27,A -85,B 0,C 180,E1 -16371.885,E2 -16371.885} C_VEL
LIN {X 0,Y 298.648,Z 175.282,A -85,B 0,C 180,E1 -16374.599,E2 -16374.599} C_VEL
LIN {X 0,Y 298.914,Z 175.25,A -85,B 0,C 180,E1 -16378.653,E2 -16378.653} C_VEL
LIN {X 0,Y 298.908,Z 175.251,A -85,B 0,C 180,E1 -16381.347,E2 -16381.347} C_VEL
LIN {X 0,Y 298.783,Z 175.269,A -85,B 0,C 180,E1 -16386.754,E2 -16386.754} C_VEL
LIN {X 0,Y 298.667,Z 175.279,A -85,B 0,C 180,E1 -16389.481,E2 -16389.481} C_VEL
LIN {X 0,Y 298.54,Z 175.295,A -85,B 0,C 180,E1 -16393.616,E2 -16393.616} C_VEL
LIN {X 0,Y 298.535,Z 175.3,A -85,B 0,C 180,E1 -16396.409,E2 -16396.409} C_VEL
LIN {X 0,Y 298.503,Z 175.3,A -85,B 0,C 180,E1 -16399.658,E2 -16399.658} C_VEL
LIN {X 0,Y 298.413,Z 175.311,A -85,B 0,C 180,E1 -16403.601,E2 -16403.601} C_VEL
LIN {X 0,Y 298.4,Z 175.313,A -85,B 0,C 180,E1 -16406.583,E2 -16406.583} C_VEL
LIN {X 0,Y 298.385,Z 175.316,A -85,B 0,C 180,E1 -16409.645,E2 -16409.645} C_VEL
LIN {X 0,Y 298.38,Z 175.314,A -85,B 0,C 180,E1 -16412.802,E2 -16412.802} C_VEL
LIN {X 0,Y 298.454,Z 175.305,A -85,B 0,C 180,E1 -16416.814,E2 -16416.814} C_VEL
LIN {X 0,Y 298.402,Z 175.313,A -85,B 0,C 180,E1 -16421.095,E2 -16421.095} C_VEL
LIN {X 0,Y 298.416,Z 175.311,A -85,B 0,C 180,E1 -16423.111,E2 -16423.111} C_VEL
LIN {X 0,Y 298.394,Z 175.314,A -85,B 0,C 180,E1 -16426.923,E2 -16426.923} C_VEL
LIN {X 0,Y 298.396,Z 175.315,A -85,B 0,C 180,E1 -16431.008,E2 -16431.008} C_VEL
LIN {X 0,Y 298.411,Z 175.311,A -85,B 0,C 180,E1 -16433.932,E2 -16433.932} C_VEL
LIN {X 0,Y 298.389,Z 175.313,A -85,B 0,C 180,E1 -16437.985,E2 -16437.985} C_VEL
LIN {X 0,Y 298.459,Z 175.305,A -85,B 0,C 180,E1 -16441.907,E2 -16441.907} C_VEL
LIN {X 0,Y 298.481,Z 175.306,A -85,B 0,C 180,E1 -16444.926,E2 -16444.926} C_VEL
LIN {X 0,Y 298.447,Z 175.307,A -85,B 0,C 180,E1 -16449.318,E2 -16449.318} C_VEL
LIN {X 0,Y 298.535,Z 175.297,A -85,B 0,C 180,E1 -16452.182,E2 -16452.182} C_VEL
LIN {X 0,Y 298.592,Z 175.289,A -85,B 0,C 180,E1 -16454.997,E2 -16454.997} C_VEL
LIN {X 0,Y 298.593,Z 175.288,A -85,B 0,C 180,E1 -16459.149,E2 -16459.149} C_VEL
LIN {X 0,Y 298.758,Z 175.27,A -85,B 0,C 180,E1 -16461.888,E2 -16461.888} C_VEL
LIN {X 0,Y 298.661,Z 175.281,A -85,B 0,C 180,E1 -16464.601,E2 -16464.601} C_VEL
LIN {X 0,Y 298.91,Z 175.25,A -85,B 0,C 180,E1 -16468.655,E2 -16468.655} C_VEL
LIN {X 0,Y 298.909,Z 175.25,A -85,B 0,C 180,E1 -16471.349,E2 -16471.349} C_VEL
LIN {X 0,Y 298.659,Z 175.281,A -85,B 0,C 180,E1 -16475.403,E2 -16475.403} C_VEL
LIN {X 0,Y 298.761,Z 175.269,A -85,B 0,C 180,E1 -16478.116,E2 -16478.116} C_VEL
LIN {X 0,Y 298.557,Z 175.293,A -85,B 0,C 180,E1 -16482.233,E2 -16482.233} C_VEL
LIN {X 0,Y 298.609,Z 175.289,A -85,B 0,C 180,E1 -16485.211,E2 -16485.211} C_VEL
LIN {X 0,Y 298.542,Z 175.299,A -85,B 0,C 180,E1 -16489.245,E2 -16489.245} C_VEL
LIN {X 0,Y 298.385,Z 175.316,A -85,B 0,C 180,E1 -16493.606,E2 -16493.606} C_VEL
LIN {X 0,Y 298.406,Z 175.313,A -85,B 0,C 180,E1 -16496.584,E2 -16496.584} C_VEL
LIN {X 0,Y 298.398,Z 175.312,A -85,B 0,C 180,E1 -16499.646,E2 -16499.646} C_VEL
LIN {X 0,Y 298.398,Z 175.317,A -85,B 0,C 180,E1 -16502.802,E2 -16502.802} C_VEL
LIN {X 0,Y 298.446,Z 175.311,A -85,B 0,C 180,E1 -16506.807,E2 -16506.807} C_VEL
LIN {X 0,Y 298.353,Z 175.32,A -85,B 0,C 180,E1 -16511.08,E2 -16511.08} C_VEL
LIN {X 0,Y 298.36,Z 175.318,A -85,B 0,C 180,E1 -16515.036,E2 -16515.036} C_VEL
LIN {X 0,Y 298.418,Z 175.311,A -85,B 0,C 180,E1 -16518.908,E2 -16518.908} C_VEL
LIN {X 0,Y 298.471,Z 175.303,A -85,B 0,C 180,E1 -16523.189,E2 -16523.189} C_VEL
LIN {X 0,Y 298.549,Z 175.4,A -85,B 0,C 180,E1 -16525.158,E2 -16525.158} C_VEL
LIN {X 0,Y 299.465,Z 180.768,A -85,B 0,C 180,E1 -16528.322,E2 -16528.322} C_VEL
LIN {X 0,Y 299.436,Z 184.576,A -85,B 0,C 180,E1 -16530.47,E2 -16530.47} C_VEL
LIN {X 0,Y 298.768,Z 191.34,A -85,B 0,C 180,E1 -16534.203,E2 -16534.203} C_VEL
LIN {X 0,Y 298.085,Z 199.35,A -85,B 0,C 180,E1 -16538.565,E2 -16538.565} C_VEL
LIN {X 0,Y 297.64,Z 205.987,A -85,B 0,C 180,E1 -16542.124,E2 -16542.124} C_VEL
LIN {X 0,Y 297.221,Z 213.935,A -85,B 0,C 180,E1 -16546.323,E2 -16546.323} C_VEL
LIN {X 0,Y 297.141,Z 216.492,A -85,B 0,C 180,E1 -16547.666,E2 -16547.666} C_VEL
LIN {X 0,Y 297.887,Z 228.641,A -85,B 0,C 180,E1 -16548.604,E2 -16548.604} C_VEL
LIN {X 0,Y 298.632,Z 237.513,A -85,B 0,C 180,E1 -16549.491,E2 -16549.491} C_VEL
LIN {X 0,Y 298.089,Z 248.255,A -85,B 0,C 180,E1 -16550.843,E2 -16550.843} C_VEL
LIN {X 0,Y 297.679,Z 256.732,A -85,B 0,C 180,E1 -16552.198,E2 -16552.198} C_VEL
LIN {X 0,Y 297.241,Z 265.455,A -85,B 0,C 180,E1 -16553.962,E2 -16553.962} C_VEL
LIN {X 0,Y 297.077,Z 271.763,A -85,B 0,C 180,E1 -16555.591,E2 -16555.591} C_VEL
LIN {X 0,Y 296.768,Z 276.892,A -85,B 0,C 180,E1 -16557.285,E2 -16557.285} C_VEL
LIN {X 0,Y 296.672,Z 280.696,A -85,B 0,C 180,E1 -16558.933,E2 -16558.933} C_VEL
LIN {X 0,Y 296.029,Z 282.655,A -85,B 0,C 180,E1 -16560.006,E2 -16560.006} C_VEL
LIN {X 0,Y 293.386,Z 285.046,A -85,B 0,C 180,E1 -16561.807,E2 -16561.807} C_VEL
LIN {X 0,Y 291.042,Z 286.482,A -85,B 0,C 180,E1 -16563.679,E2 -16563.679} C_VEL
LIN {X 0,Y 290.874,Z 286.751,A -85,B 0,C 180,E1 -16564.841,E2 -16564.841} C_VEL
LIN {X 0,Y 291.238,Z 286.821,A -85,B 0,C 180,E1 -16565.539,E2 -16565.539} C_VEL
LIN {X 0,Y 291.69,Z 286.399,A -85,B 0,C 180,E1 -16566.919,E2 -16566.919} C_VEL
LIN {X 0,Y 292.453,Z 285.364,A -85,B 0,C 180,E1 -16568.29,E2 -16568.29} C_VEL
LIN {X 0,Y 294.016,Z 282.661,A -85,B 0,C 180,E1 -16570.328,E2 -16570.328} C_VEL
LIN {X 0,Y 295.93,Z 278.549,A -85,B 0,C 180,E1 -16572.342,E2 -16572.342} C_VEL
LIN {X 0,Y 298.382,Z 272.85,A -85,B 0,C 180,E1 -16574.319,E2 -16574.319} C_VEL
LIN {X 0,Y 300.703,Z 266.748,A -85,B 0,C 180,E1 -16575.939,E2 -16575.939} C_VEL
LIN {X 0,Y 303.054,Z 259.233,A -85,B 0,C 180,E1 -16577.547,E2 -16577.547} C_VEL
LIN {X 0,Y 303.356,Z 251.427,A -85,B 0,C 180,E1 -16579.226,E2 -16579.226} C_VEL
LIN {X 0,Y 302.625,Z 243.019,A -85,B 0,C 180,E1 -16580.979,E2 -16580.979} C_VEL
LIN {X 0,Y 300.663,Z 233.223,A -85,B 0,C 180,E1 -16583.025,E2 -16583.025} C_VEL
LIN {X 0,Y 297.853,Z 223.492,A -85,B 0,C 180,E1 -16585.133,E2 -16585.133} C_VEL
LIN {X 0,Y 296.376,Z 219.851,A -85,B 0,C 180,E1 -16586.021,E2 -16586.021} C_VEL
LIN {X 0,Y 296.212,Z 218.824,A -85,B 0,C 180,E1 -16586.226,E2 -16586.226} C_VEL
LIN {X 0,Y 297.699,Z 214.954,A -85,B 0,C 180,E1 -16589.72,E2 -16589.72} C_VEL
LIN {X 0,Y 298.636,Z 212.69,A -85,B 0,C 180,E1 -16592.087,E2 -16592.087} C_VEL
LIN {X 0,Y 299.092,Z 210.813,A -85,B 0,C 180,E1 -16594.669,E2 -16594.669} C_VEL
LIN {X 0,Y 299.218,Z 209.354,A -85,B 0,C 180,E1 -16597.639,E2 -16597.639} C_VEL
LIN {X 0,Y 299.274,Z 208.444,A -85,B 0,C 180,E1 -16601.28,E2 -16601.28} C_VEL
LIN {X 0,Y 299.487,Z 208.481,A -85,B 0,C 180,E1 -16604.749,E2 -16604.749} C_VEL
LIN {X 0,Y 299.686,Z 209.067,A -85,B 0,C 180,E1 -16607.147,E2 -16607.147} C_VEL
LIN {X 0,Y 299.877,Z 209.836,A -85,B 0,C 180,E1 -16608.986,E2 -16608.986} C_VEL
LIN {X 0,Y 300.244,Z 212.135,A -85,B 0,C 180,E1 -16612.51,E2 -16612.51} C_VEL
LIN {X 0,Y 300.781,Z 215.241,A -85,B 0,C 180,E1 -16615.888,E2 -16615.888} C_VEL
LIN {X 0,Y 301.174,Z 218.087,A -85,B 0,C 180,E1 -16618.327,E2 -16618.327} C_VEL
LIN {X 0,Y 300.81,Z 220.51,A -85,B 0,C 180,E1 -16619.861,E2 -16619.861} C_VEL
LIN {X 0,Y 301.583,Z 223.553,A -85,B 0,C 180,E1 -16620.315,E2 -16620.315} C_VEL
LIN {X 0,Y 302.819,Z 227.759,A -85,B 0,C 180,E1 -16620.994,E2 -16620.994} C_VEL
LIN {X 0,Y 305.215,Z 239.265,A -85,B 0,C 180,E1 -16622.736,E2 -16622.736} C_VEL
LIN {X 0,Y 306.283,Z 248.924,A -85,B 0,C 180,E1 -16624.151,E2 -16624.151} C_VEL
LIN {X 0,Y 306.247,Z 257.528,A -85,B 0,C 180,E1 -16625.395,E2 -16625.395} C_VEL
LIN {X 0,Y 305.502,Z 262.493,A -85,B 0,C 180,E1 -16626.078,E2 -16626.078} C_VEL
LIN {X 0,Y 302.786,Z 272.298,A -85,B 0,C 180,E1 -16627.479,E2 -16627.479} C_VEL
LIN {X 0,Y 300.067,Z 281.264,A -85,B 0,C 180,E1 -16629.071,E2 -16629.071} C_VEL
LIN {X 0,Y 297.644,Z 288.745,A -85,B 0,C 180,E1 -16630.695,E2 -16630.695} C_VEL
LIN {X 0,Y 295.59,Z 295.02,A -85,B 0,C 180,E1 -16632.351,E2 -16632.351} C_VEL
LIN {X 0,Y 293.481,Z 302.13,A -85,B 0,C 180,E1 -16634.725,E2 -16634.725} C_VEL
LIN {X 0,Y 291.793,Z 306.941,A -85,B 0,C 180,E1 -16636.771,E2 -16636.771} C_VEL
LIN {X 0,Y 290.722,Z 310.677,A -85,B 0,C 180,E1 -16638.847,E2 -16638.847} C_VEL
LIN {X 0,Y 290.186,Z 312.632,A -85,B 0,C 180,E1 -16640.237,E2 -16640.237} C_VEL
LIN {X 0,Y 289.844,Z 314.136,A -85,B 0,C 180,E1 -16641.633,E2 -16641.633} C_VEL
LIN {X 0,Y 289.558,Z 315.958,A -85,B 0,C 180,E1 -16644.426,E2 -16644.426} C_VEL
LIN {X 0,Y 289.564,Z 316.236,A -85,B 0,C 180,E1 -16645.822,E2 -16645.822} C_VEL
LIN {X 0,Y 289.873,Z 315.585,A -85,B 0,C 180,E1 -16648.609,E2 -16648.609} C_VEL
LIN {X 0,Y 289.941,Z 314.587,A -85,B 0,C 180,E1 -16649.998,E2 -16649.998} C_VEL
LIN {X 0,Y 289.97,Z 313.13,A -85,B 0,C 180,E1 -16651.387,E2 -16651.387} C_VEL
LIN {X 0,Y 289.877,Z 310.025,A -85,B 0,C 180,E1 -16653.473,E2 -16653.473} C_VEL
LIN {X 0,Y 289.979,Z 305.764,A -85,B 0,C 180,E1 -16655.561,E2 -16655.561} C_VEL
LIN {X 0,Y 290.078,Z 300.113,A -85,B 0,C 180,E1 -16657.655,E2 -16657.655} C_VEL
LIN {X 0,Y 290.298,Z 292.875,A -85,B 0,C 180,E1 -16659.755,E2 -16659.755} C_VEL
LIN {X 0,Y 290.703,Z 285.402,A -85,B 0,C 180,E1 -16661.502,E2 -16661.502} C_VEL
LIN {X 0,Y 291.357,Z 275.129,A -85,B 0,C 180,E1 -16663.422,E2 -16663.422} C_VEL
LIN {X 0,Y 292.022,Z 264.536,A -85,B 0,C 180,E1 -16664.992,E2 -16664.992} C_VEL
LIN {X 0,Y 292.822,Z 253.296,A -85,B 0,C 180,E1 -16666.309,E2 -16666.309} C_VEL
LIN {X 0,Y 293.093,Z 246.105,A -85,B 0,C 180,E1 -16666.99,E2 -16666.99} C_VEL
